			IF deviceAddrIsValid
			THEN
				Busy										:= TRUE;
				Done										:= FALSE;
				Error										:= FALSE;
				ErrorId 									:= 0;
				ErrorText									:= '';
				state										:= 1001;
			ELSE
				Busy										:= FALSE;
				Done										:= FALSE;
				Error										:= TRUE;
				ErrorId 									:= 24; //Invalid ads port 
				ErrorText									:= CONCAT('Error read parameter in state:' , TO_STRING(state * -1));
				ErrorText									:= CONCAT(ErrorText , '| ID/Addr. of device invalid');
				state										:= 9999;			
			END_IF
		ELSE                        						
			Busy											:= FALSE;
			Done											:= FALSE;
			Error											:= FALSE;
			ErrorId 										:= 0;
			ErrorText										:= '';
		END_IF

	1..99,1001..1099: (* Call sequence read *)
		IF SeqRead(state)
		THEN
			state											:= 9999;	
			InitDone										:= TRUE;
			Done											:= NOT Error;
			Busy											:= FALSE;		
		END_IF
             				
	9999: (* Last state execution finished *****************************)
		IF NOT Execute 
		THEN
			Busy											:= FALSE;
			Done											:= FALSE;
			Error											:= FALSE;
			ErrorId 										:= 0;
			ErrorText										:= '';
		END_IF
		
	ELSE (* Case else *)	
		Busy												:= FALSE;
		Error												:= TRUE;
		ErrorId												:= E_AdsErr.DEVICE_INVALIDSTATE;
		ErrorText											:= CONCAT('Error read parameter; invalid state:' , TO_STRING(state));
		ErrorText											:= CONCAT(ErrorText , ' Id:');
		ErrorText											:= CONCAT(ErrorText , TO_STRING(ErrorId));
		State												:= 9999;
	END_CASE

	(* Reset state to zero if Execute is set back to false *)
	IF NOT Execute AND NOT busy
	THEN
		MemFnc												:=  -1;
		state 												:= 0;
	END_IF
	
	Read													:= Busy; //Return;
END_IF	

(****************************************************************************************************************)
END_METHOD

METHOD PROTECTED seqRead : BOOL //Return value = TRUE if execution finished 
VAR_IN_OUT
	state							:	INT;
END_VAR
CASE state OF
1,1001:
(* Example
		IF getValue(IDxGrp:= 16#5100,	IDxOffs := 16#9,	LEN := SIZEOF(uiValue),	pActValue := ADR(uiValue),  pSetValue := 0)
		THEN
			SetRefFlag :=RefFlag							:= TO_BOOL(uiValue);
		END_IF
*)
	SeqRead													:= TRUE;
ELSE
	SeqRead													:= TRUE;
END_CASE
END_METHOD

METHOD PROTECTED seqWrite : BOOL //Return value = TRUE if execution finished 
VAR_IN_OUT
	state							:	INT;
END_VAR
CASE state OF
1,1001:
(* Example 
	setValue(IDxGrp:= 16#4000,	IDxOffs := 16#102,	LEN := SIZEOF(SetDec), pActValue := ADR(Dec),	pSetValue := ADR(SetDec));
*)
	SeqWrite												:= TRUE;
ELSE
	SeqWrite												:= TRUE;
END_CASE
END_METHOD

METHOD PUBLIC FINAL write : BOOL //Return value = TRUE if busy
VAR_INPUT
	Execute													:	BOOL;
END_VAR
IF MemFnc = FNC_READ AND busy
THEN
	Busy													:= FALSE;
	Error													:= TRUE;
	ErrorId													:= E_AdsErr.DEVICE_BUSY;
	ErrorText												:= CONCAT('Error write parameter in state:' , TO_STRING(state * -1));
	ErrorText												:= CONCAT(ErrorText , ' read parameter is active, Id:');
	ErrorText												:= CONCAT(ErrorText , TO_STRING(ErrorId));
	MemFnc													:=  -1;
	Write													:= FALSE;
ELSE
	MemFnc													:= FNC_WRITE;
	THIS^.Execute											:= Execute;

(* Parameter schreiben ************************************************************************************************)
	(* Parameter schreiben Statemaschine *)
	CASE state OF
	0:	(* Init *)	
		IF Execute 
		THEN
			IF deviceAddrIsValid
			THEN
				Busy										:= TRUE;
				Done										:= FALSE;
				Error										:= FALSE;
				ErrorId 									:= 0;
				state										:= 1001;
			ELSE
				Busy										:= FALSE;
				Done										:= FALSE;
				Error										:= TRUE;
				ErrorId 									:= 24; //Invalid ads port 	
				ErrorText									:= CONCAT('Error write parameter in state:' , TO_STRING(state * -1));
				ErrorText									:= CONCAT(ErrorText , '| ID/Addr. of device invalid');
				state										:= 9999;			
			END_IF                  						
		ELSE 
			Busy											:= FALSE;
			Done											:= FALSE;
			Error											:= FALSE;
			ErrorId 										:= 0;
			ErrorText										:= '';
		END_IF
		
	1..99,1001..1099: (* Call sequence write *)
		IF SeqWrite(state)
		THEN
			Done											:= NOT Error;
			Busy											:= FALSE;
			state											:= 9999;			
		END_IF	
		
	9999: (* Last state execution finished *****************************)
		IF NOT Execute 
		THEN
			Busy											:= FALSE;
			Done											:= FALSE;
			Error											:= FALSE;
			ErrorId 										:= 0;
			ErrorText										:= '';
		END_IF
		
	ELSE (* Case else *)	
		Busy												:= FALSE;
		Error												:= TRUE;
		ErrorId												:= E_AdsErr.DEVICE_INVALIDSTATE;
		ErrorText											:= CONCAT('Error write parameter; invalid state:' , TO_STRING(state));
		ErrorText											:= CONCAT(ErrorText , ' Id:');
		ErrorText											:= CONCAT(ErrorText , TO_STRING(ErrorId));
		State												:= 9999;
	END_CASE

	(* Reset state to zero if Execute is set back to false *)
	IF NOT Execute AND NOT busy
	THEN
		MemFnc												:=  -1;
		state 												:= 0;
	END_IF
	
	Write													:= Busy; //Return;
END_IF
END_METHOD

END_FUNCTION_BLOCK

// POUs/IO/Drives/CoE/EL72xx/AxDriveCoE_wEvents
{attribute 'no_check'}
//Drive 
FUNCTION_BLOCK AxDriveCoE_wEvents EXTENDS AxDriveCoE   
VAR_OUTPUT CONSTANT
{attribute 'displaymode':='binary'}  
	OPTION_DISABLE_INT_LIMIT_WARNING						:	BYTE := 2#0000_0001;
{attribute 'displaymode':='binary'}  
	OPTION_DISABLE_REMOTE_CNTR_NOT_ACTIVE					:	BYTE := 2#0000_0010;	
END_VAR                  						
VAR_INPUT                           						
	EnableEvent												:	BOOL := TRUE;
	{attribute 'displaymode':='binary'}  
	Options													:	BYTE := 0;
	ConfirmTrig												:	BOOL := FALSE; (* Reset event *)
	SourceId												:	UDINT := 102200; //CoE Drive default multisource Id + Ax id
	Name													:	STRING(30) := '';
	ErrorLimitPos											:	BOOL := FALSE;
	ErrorLimitNeg											:	BOOL := FALSE;
END_VAR
VAR_IN_OUT
END_VAR
VAR_OUTPUT
	EventStatus												:	DWORD;
	NoOfActiveEvents										:	INT;
END_VAR                             						
VAR

END_VAR
VAR
(* Cache *********************************************************************)
	
(* Timer ********************************************************************************)
                                						
(* Trigger ******************************************************************************)


(* Function blocks ****************************************************************************)
	
	Event													: EventHandlingGrp10;
	EventDiagMessage										: EventHandling;

(* Dummy Speicher **********************************************************)
	i														: INT := 0 ;

END_VAR

	(* CoE Drive with diag and eventlogger implementation								*)
	(************************************************************************************)

(* call super ***********************************************************************)
	SUPER^();

(* trigger events ************************************************)
	_callEvents();

(*****************************************************************)

METHOD _callEvents : BOOL
VAR_INPUT
END_VAR
(* Check if msg activ and init some parameter ***********************)
	IF Event.no[1].Text2 <> Name AND Name <> '' OR Event.no[1].Text2 = '' AND rAxis.NcToPlc.AxisId <> 0
	THEN
		Event.no[1].Class 									:= TC2_SYSTEM.TCEVENTCLASS_STATEINFO;
		Event.no[3].Class 									:= TC2_SYSTEM.TCEVENTCLASS_WARNING;
		Event.no[4].Class 									:= TC2_SYSTEM.TCEVENTCLASS_WARNING;
		Event.no[5].Class 									:= TC2_SYSTEM.TCEVENTCLASS_STATEINFO;
		Event.no[6].Class 									:= TC2_SYSTEM.TCEVENTCLASS_STATEINFO;
		Event.no[7].Class 									:= TC2_SYSTEM.TCEVENTCLASS_STATEINFO;
		
		(* Init axisname *)
		FOR i := Event.MIN_EVENT TO Event.MAX_EVENT DO
		(*	Event.no[i].Text1								:= '';*)
			Event.no[i].Text2								:= SEL(LEN(name)>1,CONCAT('Axis id:',DWORD_TO_STRING(rAxis.NcToPlc.AxisId)),name);			
		END_FOR
		EventDiagMessage.Text2								:= Event.no[1].Text2;
	END_IF

(* workl Event Ctrl *************************************************)
	Event(
		ConfirmTrig 	:= ConfirmTrig,
		Disable			:= rAxis.NcToPlc.AxisId = 0 OR NOT EnableEvent,
		SourceId		:= SourceId + rAxis.NcToPlc.AxisId);
		

(* Event diag message ***************************************************)
	CASE ReadCoEDiagMsg.MsgSeverity OF
	0: // Info message
		EventDiagMessage.Class 								:= TCEVENTCLASS_MESSAGE;
	1: // warning
		EventDiagMessage.Class 								:= TCEVENTCLASS_WARNING;
	2: // error message
		EventDiagMessage.Class 								:= TCEVENTCLASS_ALARM;
	ELSE // unknown type
		EventDiagMessage.Class 								:= TCEVENTCLASS_NONE;
	END_CASE
				
	EventDiagMessage(
		Flag			:= state = 0 AND ReadCoEDiagMsg.TextId <> 0 AND (Status.Fault OR Status.Warning) AND NOT Event.Disable,
		ConfirmTrig 	:= ConfirmTrig OR NOT EventDiagMessage.Flag AND EventDiagMessage.State <> TCEVENTSTATE_INVALID,
		MsgId			:= ReadCoEDiagMsg.TextId,
		SourceId		:= Event.SourceId);
		
(* Event status ******************************************************)
	NoOfActiveEvents										:= Event.NoOfActiveEvents + SEL(EventDiagMessage.Status.31 , 0, 1);
 	EventStatus												:= Event.Status OR EventDiagMessage.Status;

		
(* Set events at the end to allow set to false in inherited FBs ********************)
	Event.no[1].Flag 										:= NOT Status.ReadyToSwitchOn; 
	Event.no[2].Flag 										:= Status.Fault;
	Event.no[3].Flag 										:= Status.Warning; 				
	Event.no[4].Flag 										:= Status.InternalLimitActive AND NOT Options.0;
	Event.no[5].Flag 										:= Status.SwitchOnDisabled;
	Event.no[6].Flag 										:= NOT Status.FollowCmdValue AND Status.SwitchedOn AND NOT options.1 AND NOT rAxis.Status.OpMode.SimulationAxis;
	Event.no[7].Flag 										:= BreakUnlock OR BreakUnlocked; 	
	Event.no[8].Flag 										:= ErrorLimitPos;
	Event.no[9].Flag 										:= ErrorLimitNeg;
	
(************************************************************************)
	_callEvents												:= TRUE;
(******************************************************************************)
END_METHOD

METHOD PUBLIC confirm : bool
VAR_INPUT
END_VAR
confirm 								:= Event.confirm();
END_METHOD

PROPERTY PUBLIC optDisabledRemoteCntrNotActive : BOOL
GET
optDisabledRemoteCntrNotActive := Options.1;
END_GET
SET
Options.1 := optDisabledRemoteCntrNotActive;
END_SET
END_PROPERTY

PROPERTY PUBLIC optDisableIntLimitWarning : BOOL
GET
optDisableIntLimitWarning := Options.0;
END_GET
SET
Options.0 := optDisableIntLimitWarning;
END_SET
END_PROPERTY

END_FUNCTION_BLOCK

// POUs/IO/Drives/CoE/CiA_DS402Controlword
FUNCTION_BLOCK CiA_DS402Controlword
VAR_INPUT

	SwitchOn 				: BOOL;	// BIT 0 
	EnableVoltage 			: BOOL := TRUE; // Bit 1 
	QuickStop 				: BOOL; // Bit 2 inverse signal / TRUE = RUN
	EnableOperation 		: BOOL; // Bit 3 
//	Operation mode specific Bit 4 	: BOOL; // Bit 4
//	Operation mode specific Bit 5 	: BOOL; // Bit 5
//	Operation mode specific Bit 6 	: BOOL; // Bit 6
	FaultReset 				: BOOL; // Bit 7 
//	Halt 					: BOOL; // Bit 8
//	Operation mode specific Bit 9 	: BOOL; // Bit 9
//	Reserved Bit 10 	: BOOL; // Bit 10
//	Manufacturere specific Bit 11 	: BOOL; // Bit 11
//	Manufacturere specific Bit 12 	: BOOL; // Bit 12
//	Manufacturere specific Bit 13 	: BOOL; // Bit 13
//	Manufacturere specific Bit 14 	: BOOL; // Bit 14
//	Manufacturere specific Bit 15 	: BOOL; // Bit 15	
END_VAR
VAR_OUTPUT
	Cmd					:	eCiA_DS402_CONTROL_CMD;
END_VAR
VAR
END_VAR

;

METHOD PUBLIC createControlword : UINT
VAR_INPUT
	StatusState												: eCiA_DS402_STATUS_STATE;
END_VAR
(* work local state machine for control ****************************************************)
	CASE StatusState OF
	eCiA_DS402_STATUS_STATE.NOT_READY_TO_SWITCH_ON:
		;
		
	eCiA_DS402_STATUS_STATE.SWITCH_ON_DISABLED:
		IF EnableVoltage
		THEN //back to "not ready to switch on"
			createControlword								:= TO_UINT(eCiA_DS402_CONTROL_CMD.SHUTDOWN);
		ELSE //To "Ready to switch on"
			createControlword								:= TO_UINT(eCiA_DS402_CONTROL_CMD.DISABLE_VOLTAGE);
		END_IF
		
	eCiA_DS402_STATUS_STATE.READY_TO_SWITCH_ON:
		IF NOT EnableVoltage
		THEN //Back to switched on disabled
			createControlword								:= TO_UINT(eCiA_DS402_CONTROL_CMD.DISABLE_VOLTAGE);
		ELSIF SwitchOn
		THEN //To switched on
			createControlword								:= TO_UINT(eCiA_DS402_CONTROL_CMD.SWITCH_ON);	
		END_IF	
		
	eCiA_DS402_STATUS_STATE.SWITCHED_ON:
		IF NOT SwitchOn
		THEN
			createControlword								:= TO_UINT(eCiA_DS402_CONTROL_CMD.SHUTDOWN);
		ELSIF NOT EnableVoltage
		THEN //Back to switched on disabled
			createControlword								:= TO_UINT(eCiA_DS402_CONTROL_CMD.DISABLE_VOLTAGE);
		ELSIF EnableOperation
		THEN // To operation enabled
			createControlword								:= TO_UINT(eCiA_DS402_CONTROL_CMD.ENABLE_OPERATION);										
		END_IF
		
	eCiA_DS402_STATUS_STATE.OPERATION_ENABLED:
		IF NOT EnableOperation 
		THEN //go back to switched on
			createControlword								:= TO_UINT(eCiA_DS402_CONTROL_CMD.SWITCH_ON);
		ELSIF NOT SwitchOn		
		THEN // back to ready to switch on 
			createControlword								:= TO_UINT(eCiA_DS402_CONTROL_CMD.SHUTDOWN);	 
		ELSIF QuickStop 
		THEN 
			createControlword								:= TO_UINT(eCiA_DS402_CONTROL_CMD.QUICK_STOP);
		ELSIF NOT EnableVoltage
		THEN //Back to switch on disabled
			createControlword								:= TO_UINT(eCiA_DS402_CONTROL_CMD.DISABLE_VOLTAGE);
		END_IF
		
	eCiA_DS402_STATUS_STATE.QUICK_STOP_ACTIVE:
		;
		
	eCiA_DS402_STATUS_STATE.FAULT_ACTIVE:
		IF NOT EnableVoltage
		THEN //back to "not ready to switch on"
			createControlword								:= TO_UINT(eCiA_DS402_CONTROL_CMD.DISABLE_VOLTAGE);
		ELSE //To "Ready to switch on"
			createControlword								:= TO_UINT(eCiA_DS402_CONTROL_CMD.SHUTDOWN);
		END_IF
		
	eCiA_DS402_STATUS_STATE.FAULT_REACTION_ACTIVE:
		;		
	END_CASE
	
(* Write controlword ********************************************************)
	Cmd													:= TO_INT(createControlword);
	createControlword.7										:= FaultReset; 
	
(*****************************************************************************)
END_METHOD

END_FUNCTION_BLOCK

// POUs/IO/Drives/DC/Ey73xx/AxDriveDC
{attribute 'no_check'}
//Beckhoff Stepper terminal status and diagnoses/ EP Box used with NC axis
//EventHandling instance use inside
FUNCTION_BLOCK AxDriveDC EXTENDS AxDriveBase
VAR CONSTANT         	
END_VAR  
VAR_INPUT
END_VAR                     					
VAR_IN_OUT                  					
END_VAR                     					
VAR_OUTPUT                  					
	Status_ReadyToEnable									: BOOL;
	Status_Ready											: BOOL;
	Status_Warning											: BOOL;
	Status_Error											: BOOL;
	Status_MovingPos										: BOOL;
	Status_MovingNeg										: BOOL;
	Status_TorqueReduced									: BOOL;
	Status_DigInput1										: BOOL;
	Status_DigInput2										: BOOL;
	Status_SyncError										: BOOL;
	Status_TxPDOToggle										: BOOL;
	InfoData1										AT %I*	:	UINT;
	InfoData2										AT %I*	:	UINT;
END_VAR                     					                   					
VAR                         					
END_VAR
VAR

(* Cache *********************************************************************)
	StatusTrig												:	BYTE;
	MemStatusTrig											:	BYTE;
	MemCoeCache												: 	ARRAY[0..5] OF BYTE; //Index A020/A030 with a lenght of 17 subindex	
	
//Diag read by CoE
	Diag_Saturated											: BOOL; // Driver stage operates with maximum duty cycle
	Diag_OverTemperature 									: BOOL; // Internal terminal temperature is higher than 80°C (see subindex 0xF80F:04)
	Diag_TorqueOverloaded 									: BOOL; // Motor current is higher than the rated current
	Diag_UnderVoltage 										: BOOL; // Motor supply voltage is 20% lower than the configured nominal voltage
	Diag_OverVoltage 										: BOOL; // Motor supply voltage is 10% higher than the configured nominal voltage
	Diag_ShortCircuit 										: BOOL; // Short circuit 
	Diag_ShortCircuitB										: BOOL; // Short circuit
	Diag_NoControlPower 									: BOOL; // Control voltage at the power contacts is less than 12 V
	Diag_MiscError 											: BOOL; // Terminal initialization failed, or supply voltage is less than 8 V, or internal terminal temperature is higher than 100°C (see subindex 0xF80F:05)
	Diag_Configuration 										: BOOL; // CoE change has not yet been adopted into the current configuration
	Diag_MotorStall											: BOOL; // A loss of step has occurred
	Diag_OpenLoadA											: BOOL; // Open load on coil A - e.g. no motor connected
	Diag_OpenLoadB											: BOOL; // Open load on coil B - e.g. no motor connected

	Diag_ActualMode											: BYTE; // Current operating mode (relevant for activated automatic mode, see 0x8012:01)
	
(* Timer ********************************************************************************)

(* Trigger ******************************************************************************)

(* Instance ****************************************************************************)
	CoERead													:	FB_EcCoeSdoReadEx := (tTimeout := DEFAULT_ADS_TIMEOUT);	//Read data via CoE
	
(* Dummy Speicher **********************************************************)
END_VAR

	(* DC Drive Control															*)
	(************************************************************************************)

(* abort function-call if the reference is invalid *****************************)
IF NOT __ISVALIDREF(rAxis) 
THEN
	Fault													:= TRUE;
	SwitchedOn												:= FALSE;
	Ready													:= FALSE;
	RETURN;
END_IF

(* Call super class ****************************************************)
	SUPER^(); 

(* Read Statusword ********************************************************)
	Status_ReadyToEnable									:= StatusWord.0 OR rAxis.Status.OpMode.SimulationAxis ;
	Status_Ready											:= StatusWord.1 OR rAxis.Status.OpMode.SimulationAxis;
	Status_Warning											:= StatusWord.2;
	Status_Error											:= StatusWord.3;
	Status_MovingPos										:= StatusWord.4;
	Status_MovingNeg										:= StatusWord.5;
	Status_TorqueReduced									:= StatusWord.6;              
             					   
	Status_DigInput1										:= StatusWord.11;
	Status_DigInput2										:= StatusWord.12;
	Status_SyncError										:= StatusWord.13;
//	_StatusWord.14;//6                                         
	Status_TxPDOToggle										:= StatusWord.15;

(* Read diag data ************************************************)
	StatusTrig.0											:= NOT Status_ReadyToEnable;
	StatusTrig.1											:= Status_Error;
	StatusTrig.2											:= Status_Warning;
	
	CASE state OF
	0:
		IF StatusTrig <> MemStatusTrig AND NOT rAxis.Status.OpMode.SimulationAxis AND AdsAddr.port > 0 
		THEN
			CoERead(
				sNetId		:= F_CreateAmsNetId(nIds :=AdsAddr.netId), 
				nSlaveAddr	:= AdsAddr.port, 
				nSubIndex	:= , 
				nIndex		:= , 
				pDstBuf		:= , 
				cbBufLen	:= , 
				bExecute	:= FALSE,
				bCompleteAccess:= TRUE, 
				tTimeout	:= , 
				bBusy		=> , 
				bError		=> , 
				nErrId		=> );
			IF NOT CoERead.bBusy
			THEN
				MemStatusTrig 								:= StatusTrig;			
				state 										:= state + 1;
			END_IF
		END_IF
	1: 
		CoERead(
			bExecute	:= TRUE, 
			nIndex		:= SEL(Channel=0,16#A030,16#A020),
			nSubIndex	:= 16#0, 
			pDstBuf		:= ADR(MemCoeCache), 
			cbBufLen	:= SIZEOF(MemCoeCache));
		IF NOT CoERead.bBusy
		THEN
			IF CoERead.bError
			THEN
				state 										:= 0;
			ELSE
				//											:= MemCoeChache[0]; 	//Subindex 0x00 Maximal sub index
				//											:= MemCoeChache[1];		//reserved				
				Diag_Saturated								:= MemCoeCache[2].0; 	//Subindex 0x01 
				Diag_OverTemperature 						:= MemCoeCache[2].1; 	//Subindex 0x02 
				Diag_TorqueOverloaded 						:= MemCoeCache[2].2; 	//Subindex 0x03 
				Diag_UnderVoltage 							:= MemCoeCache[2].3; 	//Subindex 0x04 
				Diag_OverVoltage 							:= MemCoeCache[2].4; 	//Subindex 0x05 
				Diag_ShortCircuit 							:= MemCoeCache[2].5; 	//Subindex 0x06   
				Diag_NoControlPower 						:= MemCoeCache[2].7; 	//Subindex 0x08 
				Diag_MiscError 								:= MemCoeCache[3].0; 	//Subindex 0x09
				Diag_Configuration 							:= MemCoeCache[3].1; 	//Subindex 0x0A
				//											:= MemCoeCache[3].2; 	//Subindex 0x0B 
				//											:= MemCoeCache[3].3; 	//Subindex 0x0C 
				//	 										:= MemCoeCache[3].4; 	//Subindex 0x0D 
				//				 							:= MemCoeChache[3].5; 	//Subindex 0x0E 
				//				 							:= MemCoeChache[3].6; 	//Subindex 0x0F 
				//				 							:= MemCoeChache[3].7; 	//Subindex 0x10 								
				Diag_ActualMode	 							:= MemCoeCache[4]; 	//Subindex 0x11 (e.g. 17) 
				//				 							:= MemCoeChache[5];		//reserved
	
				state										:= 0;			
			END_IF
			CoERead(bExecute := False);		
		END_IF
	END_CASE
	
(* DriveStatusBits ***********************************************)
	Fault													:= Status_Error
															//	OR Status_MotorStall
																OR Status_SyncError
																OR rAxis.NcToPlc.StateDWord.28 (* DriveDeviceError *)
																OR rAxis.NcToPlc.StateDWord.30; (* IODataInvalid *)
         											
													
	Ready	 												:= NOT Fault
																AND(Status_ReadyToEnable OR Status_Ready);
	SwitchedOn												:= Status_Ready AND NOT Fault;
	
(*******************************************************************)

END_FUNCTION_BLOCK

// POUs/IO/Drives/DC/Ey73xx/AxDriveDC_wEvents
{attribute 'no_check'}
//Beckhoff Stepper terminal diag and diagnosis with eventlogger - extended from AxDriveStepper
//EventHandling instance use inside
FUNCTION_BLOCK AxDriveDC_wEvents EXTENDS AxDriveDC
VAR CONSTANT         	
END_VAR  
VAR_INPUT
	EnableEvent												:	BOOL := TRUE; //Enable to show events
	ConfirmTrig												:	BOOL := FALSE; //Quit events
	SourceId												:	UDINT := 102700; //CoE / MDP733 DC-Motor Drive (EL73xx) default multisource Id + Ax id
	Name													:	STRING(30) := '';
	ErrorLimitPos											:	BOOL := FALSE;
	ErrorLimitNeg											:	BOOL := FALSE;
END_VAR                     					
VAR_IN_OUT                  					
END_VAR                     					
VAR_OUTPUT                  					
 	EventStatus												:	DWORD;       
	NoOfActiveEvents										:	INT;                    					
END_VAR                     					                   					
VAR                         					
END_VAR
VAR

(* Cache *********************************************************************)
	
(* Timer ********************************************************************************)

(* Trigger ******************************************************************************)

(* Instance ****************************************************************************)
	Event													:	EventHandlingGrp10;
	
(* Dummy Speicher **********************************************************)
	i														: INT := 0 ;
END_VAR

	(* Stepper Drive Control with events												*)
	(************************************************************************************)

(* Call super **********************************************)
	SUPER^();
	
(* work events *******************************************)
	_callEvents();

(*******************************************************)

METHOD PRIVATE _callEvents : BOOL
VAR_INPUT
END_VAR

(* Check if msg activ and init some parameter ***********************)
	IF Event.no[1].Text2 <> Name AND Name <> '' OR Event.no[1].Text2 = '' AND rAxis.NcToPlc.AxisId <> 0
	THEN
		Event.no[1].Class 									:= TC2_SYSTEM.TCEVENTCLASS_STATEINFO;
		Event.no[3].Class 									:= TC2_SYSTEM.TCEVENTCLASS_WARNING;
		
		(* Init Achsname *)
		FOR i := Event.MIN_EVENT TO Event.MAX_EVENT DO
		(*	Event.no[i].Text1								:= '';*)
			Event.no[i].Text2								:= SEL(LEN(name)>1,CONCAT('Axis id:',DWORD_TO_STRING(rAxis.NcToPlc.AxisId)),name);
		END_FOR
	END_IF

(* workl Event Ctrl *************************************************)
	Event(
		ConfirmTrig := ConfirmTrig,
		Disable		:= rAxis.NcToPlc.AxisId = 0 OR NOT EnableEvent,
		SourceId	:= SourceId + rAxis.NcToPlc.AxisId,
		Status		=> EventStatus,
		NoOfActiveEvents => NoOfActiveEvents);

(* Event Logger Meldungen *****************************************************)
	Event.no[1].Flag 										:= NOT Status_ReadyToEnable ; 
	Event.no[2].Flag 										:= Fault;
	Event.no[3].Flag 										:= (Status_Warning OR Diag_Configuration) AND NOT rAxis.Status.Homing AND NOT rAxis.Status.Disabled; //Avoid warning if drive is disabled (EL7037 and older FB on EL7047 - 2020-03-26) 				
	Event.no[4].Flag 										:= Diag_TorqueOverloaded;
	Event.no[5].Flag 										:= Diag_UnderVoltage OR Diag_OverVoltage OR Diag_NoControlPower;
	Event.no[6].Flag 										:= Diag_ShortCircuit;
	Event.no[7].Flag 										:= Diag_Saturated;
	Event.no[8].Flag										:= Diag_OverTemperature ;
	Event.no[9].Flag 										:= ErrorLimitPos; 	
	Event.no[10].Flag 										:= ErrorLimitNeg;	
(*	Event.no[11].Flag 										:= FALSE; 				
	Event.no[12].Flag 										:= FALSE;					
	Event.no[13].Flag 										:= FALSE; 			Event.no[9].Class := TC2_SYSTEM.TCEVENTCLASS_WARNING;
	Event.no[14].Flag 										:= FALSE; 			Event.no[10].Class := TC2_SYSTEM.TCEVENTCLASS_WARNING;
	Event.no[15].Flag 										:= FALSE;
	Event.no[16].Flag 										:= FALSE;
	Event.no[17].Flag 										:= FALSE;
	Event.no[18].Flag 										:= FALSE;
	Event.no[19].Flag 										:= FALSE;
	Event.no[20].Flag 										:= FALSE;
	Event.no[21].Flag 										:= FALSE;
	Event.no[22].Flag 										:= FALSE;
	Event.no[23].Flag 										:= FALSE;
	Event.no[24].Flag 										:= FALSE;
	Event.no[25].Flag 										:= FALSE;
*)

(******************************************************************************)
END_METHOD

METHOD PUBLIC confirm : bool
VAR_INPUT
END_VAR
confirm			:= Event.confirm();
END_METHOD

END_FUNCTION_BLOCK

// POUs/IO/Drives/Stepper/AxDriveStepper
{attribute 'no_check'}
//Beckhoff Stepper terminal status and diagnoses/ EP Box used with NC axis
//EventHandling instance use inside
FUNCTION_BLOCK AxDriveStepper EXTENDS AxDriveBase
VAR CONSTANT         	
END_VAR  
VAR_INPUT
END_VAR                     					
VAR_IN_OUT                  					
END_VAR                     					
VAR_OUTPUT                  					
	Status_ReadyToEnable									: BOOL;
	Status_Ready											: BOOL;
	Status_Warning											: BOOL;
	Status_Error											: BOOL;
	Status_MovingPos										: BOOL;
	Status_MovingNeg										: BOOL;
	Status_TorqueReduced									: BOOL;
	Status_MotorStall										: BOOL;
	Status_DigInput1										: BOOL;
	Status_DigInput2										: BOOL;
	Status_SyncError										: BOOL;
	Status_TxPDOToggle										: BOOL;
	InfoData1										AT %I*	:	UINT;
	InfoData2										AT %I*	:	UINT;
END_VAR                     					                   					
VAR                         					
END_VAR
VAR

(* Cache *********************************************************************)
	StatusTrig												:	BYTE;
	MemStatusTrig											:	BYTE;
	MemCoeCache											: 	ARRAY[0..5] OF BYTE; //Index A010 with a lenght of 17 subindex	
	
//Diag read by CoE
	Diag_Saturated											: BOOL; // Driver stage operates with maximum duty cycle
	Diag_OverTemperature 									: BOOL; // Internal terminal temperature is higher than 80°C (see subindex 0xF80F:04)
	Diag_TorqueOverloaded 									: BOOL; // Motor current is higher than the rated current
	Diag_UnderVoltage 										: BOOL; // Motor supply voltage is 20% lower than the configured nominal voltage
	Diag_OverVoltage 										: BOOL; // Motor supply voltage is 10% higher than the configured nominal voltage
	Diag_ShortCircuit 										: BOOL; // Short circuit 
	Diag_ShortCircuitB										: BOOL; // Short circuit
	Diag_NoControlPower 									: BOOL; // Control voltage at the power contacts is less than 12 V
	Diag_MiscError 											: BOOL; // Terminal initialization failed, or supply voltage is less than 8 V, or internal terminal temperature is higher than 100°C (see subindex 0xF80F:05)
	Diag_Configuration 										: BOOL; // CoE change has not yet been adopted into the current configuration
	Diag_MotorStall											: BOOL; // A loss of step has occurred
	Diag_OpenLoadA											: BOOL; // Open load on coil A - e.g. no motor connected
	Diag_OpenLoadB											: BOOL; // Open load on coil B - e.g. no motor connected

	Diag_ActualMode											: BYTE; // Current operating mode (relevant for activated automatic mode, see 0x8012:01)
	
(* Timer ********************************************************************************)

(* Trigger ******************************************************************************)

(* Instance ****************************************************************************)
	CoERead													:	FB_EcCoeSdoReadEx := (tTimeout := DEFAULT_ADS_TIMEOUT);	//Read data via CoE
	
(* Dummy Speicher **********************************************************)
END_VAR

	(* Stepper Drive Control															*)
	(************************************************************************************)

(* abort function-call if the reference is invalid *****************************)
IF NOT __ISVALIDREF(rAxis) 
THEN
	Fault													:= TRUE;
	SwitchedOn												:= FALSE;
	Ready													:= FALSE;
	RETURN;
END_IF

(* Call super class ****************************************************)
	SUPER^();
	
(* Read Statusword ********************************************************)
	Status_ReadyToEnable									:= StatusWord.0 OR rAxis.Status.OpMode.SimulationAxis ;
	Status_Ready											:= StatusWord.1 OR rAxis.Status.OpMode.SimulationAxis;
	Status_Warning											:= StatusWord.2;
	Status_Error											:= StatusWord.3;
	Status_MovingPos										:= StatusWord.4;
	Status_MovingNeg										:= StatusWord.5;
	Status_TorqueReduced									:= StatusWord.6;
	Status_MotorStall										:= StatusWord.7;
//	_StatusWord.8; //0                  					   
//	_StatusWord.9; //1                  					   
//	_StatusWord.10;//2                  					   
	Status_DigInput1										:= StatusWord.11;
	Status_DigInput2										:= StatusWord.12;
	Status_SyncError										:= StatusWord.13;
//	_StatusWord.14;//6                                         
	Status_TxPDOToggle										:= StatusWord.15;

(* Read diag data ************************************************)
	StatusTrig.0											:= NOT Status_ReadyToEnable;
	StatusTrig.1											:= Status_Error;
	StatusTrig.2											:= Status_Warning;
	
	CASE state OF
	0:
		IF StatusTrig <> MemStatusTrig AND NOT rAxis.Status.OpMode.SimulationAxis AND AdsAddr.port > 0 
		THEN
			CoERead(
				sNetId		:= F_CreateAmsNetId(nIds :=AdsAddr.netId), 
				nSlaveAddr	:= AdsAddr.port, 
				nSubIndex	:= , 
				nIndex		:= , 
				pDstBuf		:= , 
				cbBufLen	:= , 
				bExecute	:= FALSE,
				bCompleteAccess:= TRUE, 
				tTimeout	:= , 
				bBusy		=> , 
				bError		=> , 
				nErrId		=> );
			IF NOT CoERead.bBusy
			THEN
				MemStatusTrig 								:= StatusTrig;			
				state 										:= state + 1;
			END_IF
		END_IF
	1: 
		CoERead(
			bExecute	:= TRUE, 
			nIndex		:= 16#A010,
			nSubIndex	:= 16#0, 
			pDstBuf		:= ADR(MemCoeCache), 
			cbBufLen	:= SIZEOF(MemCoeCache));
		IF NOT CoERead.bBusy
		THEN
			IF CoERead.bError
			THEN
				state 										:= 0;
			ELSE
				//											:= MemCoeChache[0]; 	//Subindex 0x00 Maximal sub index
				//											:= MemCoeChache[1];		//reserved				
				Diag_Saturated								:= MemCoeCache[2].0; 	//Subindex 0x01 
				Diag_OverTemperature 						:= MemCoeCache[2].1; 	//Subindex 0x02 
				Diag_TorqueOverloaded 						:= MemCoeCache[2].2; 	//Subindex 0x03 
				Diag_UnderVoltage 							:= MemCoeCache[2].3; 	//Subindex 0x04 
				Diag_OverVoltage 							:= MemCoeCache[2].4; 	//Subindex 0x05 
				Diag_ShortCircuit 							:= MemCoeCache[2].5; 	//Subindex 0x06   
				Diag_ShortCircuitB 							:= MemCoeCache[2].6; 	//Subindex 0x07 - only at EL70x1
				Diag_NoControlPower 						:= MemCoeCache[2].7; 	//Subindex 0x08 
				Diag_MiscError 								:= MemCoeCache[3].0; 	//Subindex 0x09
				Diag_Configuration 							:= MemCoeCache[3].1; 	//Subindex 0x0A
				Diag_MotorStall 							:= MemCoeCache[3].2; 	//Subindex 0x0B 
				Diag_OpenLoadA 								:= MemCoeCache[3].3; 	//Subindex 0x0C 
				Diag_OpenLoadB	 							:= MemCoeCache[3].4; 	//Subindex 0x0D 
				//				 							:= MemCoeChache[3].5; 	//Subindex 0x0E 
				//				 							:= MemCoeChache[3].6; 	//Subindex 0x0F 
				//				 							:= MemCoeChache[3].7; 	//Subindex 0x10 								
				Diag_ActualMode	 							:= MemCoeCache[4]; 	//Subindex 0x11 (e.g. 17) 
				//				 							:= MemCoeChache[5];		//reserved
	
				state										:= 0;			
			END_IF
			CoERead(bExecute := False);		
		END_IF
	END_CASE
	
(* DriveStatusBits ***********************************************)
	Fault													:= Status_Error
															//	OR Status_MotorStall
																OR Status_SyncError
																OR rAxis.NcToPlc.StateDWord.28 (* DriveDeviceError *)
																OR rAxis.NcToPlc.StateDWord.30; (* IODataInvalid *)
         											
													
	Ready	 												:= NOT Fault
																AND(Status_ReadyToEnable OR Status_Ready);
	SwitchedOn												:= Status_Ready AND NOT Fault;
	
(*******************************************************************)

END_FUNCTION_BLOCK

// POUs/IO/Drives/SoE/Ax580x
{attribute 'no_check'}
//AX5000 safety card option IOs - AX5805/AX5806 FSoE slave inputs 
FUNCTION_BLOCK Ax580x 
VAR_INPUT
END_VAR
VAR_OUTPUT
	STO												AT %I*		:	BOOL;	//option Safe Torque Off
	SSM_1											AT %I*		:	BOOL;	//option Safe Speed Monitor 1
	SSM_2											AT %I*		:	BOOL;	//option Safe Speed Monitor 2
	SOS_1											AT %I*		:	BOOL;	//option Safe Operating Speed 1
	SSR_1											AT %I*		:	BOOL;	//option Safe Speed Range 1
	SDIp											AT %I*		:	BOOL;	//option Safe Direction positive
	SDIn											AT %I*		:	BOOL;	//option Safe Direction negative
	Error											AT %I*		:	BOOL;	//Error active or error ack 
	SLS_1											AT %I*		:	BOOL;	//special config (Safe Limited Speed)
	
	PositionActualValue								AT %I*	:	DINT;		//contains actual position value of drive 
	VelocityActualValue								AT %I*	:	DINT;		//contains actual velocity value of drive	
END_VAR         								
VAR             								
END_VAR

(* AX5805/06 AX5000 servo drives safety card FSoE slave inputs		*)
(********************************************************************)

(* Input Signals Valid ******************************************************)
(* not in use
	STO														:= SafeDataByte.0;
	SSM_1													:= SafeDataByte.1;
	SSM_2													:= SafeDataByte.2;
	SOS_1													:= SafeDataByte.3;
	SSR_1													:= SafeDataByte.4;
	SDIp													:= SafeDataByte.5;
	SDIn													:= SafeDataByte.6;
	Error													:= SafeDataByte.7;
	SLS_1													:= SafeDataByte.8; // Special Config
*)
(**********************************************************************)

END_FUNCTION_BLOCK

// POUs/IO/Drives/SoE/AxDriveSoE_Ax5000
{attribute 'no_check'}
//AX5000 SoE drive status and diagnosis FB
FUNCTION_BLOCK AxDriveSoE_Ax5000 extends AxDriveBase (* Lips: TcMc2Drive, TcDrive *)
VAR_INPUT
	ResetTrig												:	BOOL;
	BreakUnlock												:	BOOL;
	BreakLock												:	BOOL;					
END_VAR                 									
VAR_IN_OUT              									
END_VAR                 									
VAR_OUTPUT              	                    										
	BreakStatus												:	BOOL; (* FALSE = ON / TRUE = OFF *)                        								
	RT_StatusChanged										:	BOOL;
{attribute 'displaymode':='binary'}
	MotorsStatusWord										:	WORD; 
	Status													:	ST_AX5000DriveStatus;
	C1D														:	ST_AX5000_C1D;
	DiagMsg 												: 	ST_SoE_String;
	DiagNumber 												: 	UDINT;
	SafetyError										AT %I*	:	BOOL;	(* Ax5805 Drive Safety Error - Bit .7 in Input Safe Data Byte 0 oder 2 *)	
	SercosErrorId											:	UINT;
END_VAR
VAR_OUTPUT CONSTANT
END_VAR
VAR (* EA Internal *)
	(* P-0-0205 - muss ins Zyklische Interface des Reglers unter S-0-0016 (AT) gemappt,
		und dann direkt mit der PLC-Variable verknüpft werden. 
		Oder für das Lesen auf Anforderung die Deklaration auf Lokale Variable ändern 
		und in der Statemaschine für das Status lesen 
		den Auskommentierten Teil mit ins Programm nehmen 
	*)
(*	PwrMgmStatusWord AT %I* : WORD; *)
(*	PwrMgmStatusWord : WORD; *)

END_VAR
VAR

(* Zwischenspeicher *********************************************************************)
	MemDriveStatusword										: 	WORD;
	
	MEM_StatusTrig											:	BYTE;
	StatusTrig												:	BYTE;
	stateReadStatus											:	INT;

(* Timer ********************************************************************************)

(* Trigger ******************************************************************************)

(* Bausteine ****************************************************************************)
	SoEAX5000SetMotorCtrlWord 								: FB_SoEAX5000SetMotorCtrlWord_ByDriveRef := (tTimeout := DEFAULT_ADS_TIMEOUT);	(* Bremse manuell lösen *)
	SoEDriveReset											: FB_SoEReset_ByDriveRef := (tTimeout	:= DEFAULT_ADS_TIMEOUT);
	SoERead													: FB_SoERead_ByDriveRef := (tTimeout:= DEFAULT_ADS_TIMEOUT);

(* Dummy Speicher **********************************************************)
	_WORD													: WORD;
(****************************************************************************)
END_VAR

	(************************************************************************************)
	(*																					*)
	(*		B E C K H O F F   N E W   A U T O M A T I O N   T E C H N O L O G Y    		*)
	(*																					*)
	(*		Eiserstr.5	D-33415 Verl	Germany	phone:	+49-5246-0	www.Beckhoff.Com	*)
    (*																					*)
    (*		Bausteinbeschreibung	:	AX5000 Drive Ctrl								*)
	(*		TwinCAT-Version			:	3.x or higher 									*)
	(*		Version					:	V3.0 											*)
 	(*		Autor					:	Daniel Schlingmann								*)
	(*		Lib						:	TcMc2Drive.lib / TcDrive.Lib					*)
	(*																					*)
	(************************************************************************************)

(* abort function-call if the reference is invalid *****************************)
IF NOT __ISVALIDREF(rAxis)  THEN
	Fault													:= TRUE;
	Ready													:= FALSE;
	SwitchedOn												:= FALSE;
	RETURN;
END_IF

(* Call super class ****************************************************)
	SUPER^(); 
	
(* DriveStatusword *****************************)
	Status 													:= F_ConvWordToSTAX5000DriveStatus(StatusWord);
	IF rAxis.Status.OpMode.SimulationAxis OR AdsAddr.port = 0
	THEN
		Status.bNotReadyToPowerUp							:= FALSE;	
		Status.bDrvShutdownBitC1D							:= FALSE;
		Status.bReadyForEnable								:= TRUE;
		Status.bEnabled										:= TRUE;	
	END_IF
	(* PowerManagementStatusWord Auswerten *)
	(* Bit 0 = Status UMain ok, ok = True
		Bit 1 = Umain Overvoltage, active = True
		Bit 2 = Umain phase error, error = False
		Bit 3 = Status DcLink ok, ok = True
		Bit 4 = Ext. Umain relay, ready to Switch on = True
		Bit 5 = Status Fan, aktive = True 
		Bit 6 = Status load relay, active = True
		Bit 7 = Status internal chopper, active = True
		Bit 8 = Status external chopper, active = True
		Bit 9 = Status additinal fan, active = True
		Bit 10-15 = reserved *)
	(*
	ReadyForContactor := PowerManagementStatusWord.4;
	*)

(* DriveStatusBits ***********************************************)
	Fault													:= Status.bDrvShutdownBitC1D
																OR rAxis.NcToPlc.StateDWord.28 (* DriveDeviceError *)
																OR rAxis.NcToPlc.StateDWord.30 (* IODataInvalid *)
																OR SafetyError;
            												
	Ready 													:= NOT Fault
																AND(Status.bReadyForEnable OR Status.bEnabled)
																(* AND ReadyForContactor AX 5000 *);

	SwitchedOn												:= Status.bEnabled AND NOT Fault;	
																
(* Init drive ref *************************************************)
	IF AdsAddr.port <> SoEDriveReset.stDriveRef.nSlaveAddr 
	THEN
		SoEDriveReset.stDriveRef.sNetId						:= F_CreateAmsNetId(AdsAddr.netId);	
		SoEDriveReset.stDriveRef.nSlaveAddr					:= AdsAddr.port;	
		SoEDriveReset.stDriveRef.nDriveNo					:= Channel;	
		
		SoEAX5000SetMotorCtrlWord.stDriveRef				:= 	
		SoERead.stDriveRef		 							:= SoEDriveReset.stDriveRef;
	END_IF

(* Reset Drive ****************************************************)
	SoEDriveReset();
	IF SoEDriveReset.bBusy 
	THEN
		; (* Block ist currend working *)
	ELSIF ResetTrig
	THEN
		reset();
	ELSIF SoEDriveReset.bExecute
	THEN
		RefreshStatus();
		SoEDriveReset.bExecute 								:= FALSE;
	END_IF

(* Bremse loesen/setzen  ***********************************************)
	IF (SoEAX5000SetMotorCtrlWord.bForceUnLock XOR BreakUnlock)
		OR (SoEAX5000SetMotorCtrlWord.bForceLock XOR Breaklock)
		OR SoEAX5000SetMotorCtrlWord.bBusy 
	THEN
		SoEAX5000SetMotorCtrlWord(
			stDriveRef	:= ,  //See above
			bExecute	:= NOT SoEAX5000SetMotorCtrlWord.bBusy AND NOT rAxis.Status.OpMode.SimulationAxis, 
			tTimeout	:= , 
			bForceLock	:= Breaklock , 
			bForceUnlock:= BreakUnlock , 
			bBusy		=> , 
			bError		=>  , 
			iAdsErrId	=> , 
			iSercosErrId=> );
	END_IF

(* DriveStatusword auswerten Sercos *****************************)
	RT_StatusChanged 										:= SHR(StatusWord,2) <> MemDriveStatusword;
	MemDriveStatusword 										:= SHR(StatusWord,2);

(* Start Read Drive status *****************************************************************)
	CASE stateReadStatus OF
	0:
		StatusTrig.0 										:= rAxis.NcToPlc.StateDWord.28;
		StatusTrig.1 										:= rAxis.NcToPlc.StateDWord.30;

		IF NOT rAxis.Status.OpMode.SimulationAxis AND AdsAddr.port > 0
			AND(RT_StatusChanged OR MEM_StatusTrig <> StatusTrig)
		THEN
			RefreshStatus();
		ELSE
			;
		END_IF

	(* Read Class 1 Diag *********************************************************)
	10:
		IF NOT SoERead.bBusy
			AND SoERead.bExecute
		THEN
			IF SoERead.bError THEN
				stateReadStatus 							:= 0;
			ELSE                        					
				C1D 										:= F_ConvWordToSTAX5000C1D(_WORD);
				stateReadStatus 							:= stateReadStatus + 1;
			END_IF
		END_IF

		SoERead(
			stDriveRef	:= ,  //See init for drive ref
			nIdn		:= S_0_IDN + 11,
			nElement	:= EC_SOE_ELEMENT_VALUE (* 16#40*),
			pDstBuf		:= ADR(_WORD),
			cbBufLen	:= SIZEOF(_WORD),
			bExecute	:= stateReadStatus = 10,
			tTimeout	:= ,
			bBusy		=> ,
			bError		=> ,
			iAdsErrId	=> ,
			iSercosErrId=> ,
			dwAttribute	=> );

	(* Motor Statusword ***************************************************)
	11:
		IF NOT SoERead.bBusy
			AND SoERead.bExecute
		THEN
			IF SoERead.bError 
			THEN
				stateReadStatus 							:= 0;
			ELSE
				BreakStatus 								:= MotorsStatusWord.0;
				stateReadStatus 							:= stateReadStatus + 1;
			END_IF
		END_IF

		SoERead(
			stDriveRef	:= ,  //See init for drive ref
			nIdn		:= P_0_IDN + 97, (* Motor Status word *)
			nElement	:= EC_SOE_ELEMENT_VALUE (* 16#40*),
			pDstBuf		:= ADR(MotorsStatusWord),
			cbBufLen	:= SIZEOF(MotorsStatusWord),
			bExecute	:= stateReadStatus = 11,
			tTimeout	:= ,
			bBusy		=> ,
			bError		=> ,
			iAdsErrId	=> ,
			iSercosErrId=> ,
			dwAttribute	=> );


	(* Diag Message *********************************************************)
	12:
		IF NOT SoERead.bBusy
			AND SoERead.bExecute
		THEN
			IF SoERead.bError 
			THEN
				stateReadStatus 							:= 0;
			ELSE
				stateReadStatus 							:= stateReadStatus + 1;
			END_IF
		END_IF

		SoERead(
			stDriveRef	:= ,  //See init for drive ref
			nIdn		:= S_0_IDN + 95,
			nElement	:= EC_SOE_ELEMENT_VALUE (* 16#40*),
			pDstBuf		:= ADR(DiagMsg),
			cbBufLen	:= SIZEOF(DiagMsg),
			bExecute	:= stateReadStatus = 12,
			tTimeout	:= ,
			bBusy		=> ,
			bError		=> ,
			iAdsErrId	=> ,
			iSercosErrId=> ,
			dwAttribute	=> );

	(* Diag Number *********************************************************)
	13:
		IF NOT SoERead.bBusy
			AND SoERead.bExecute
		THEN
			IF SoERead.bError 
			THEN
				stateReadStatus 							:= 0;
			ELSE
				stateReadStatus 							:= stateReadStatus + 1;
			END_IF
		END_IF
		
		SoERead(
			stDriveRef	:= ,  //See init for drive ref
			nIdn		:= S_0_IDN + 390,
			nElement	:= EC_SOE_ELEMENT_VALUE (* 16#40*),
			pDstBuf		:= ADR(DiagNumber),
			cbBufLen	:= SIZEOF(DiagNumber),
			bExecute	:= stateReadStatus = 13,
			tTimeout	:= ,
			bBusy		=> ,
			bError		=> ,
			iAdsErrId	=> ,
			iSercosErrId=> ,
			dwAttribute	=> );

	(* reading status finished ************************************************************)
	ELSE (* Case else *)
		stateReadStatus 									:= 0;
	END_CASE

(******************************************************************************************)

METHOD PUBLIC break : BOOL //Return value = TRUE if busy
VAR_INPUT
	lock													: BOOL;
END_VAR
BreakLock													:= lock AND NOT rAxis.Status.OpMode.SimulationAxis;
BreakUnlock													:= NOT lock AND NOT rAxis.Status.OpMode.SimulationAxis;
break														:= (SoEAX5000SetMotorCtrlWord.bForceUnLock XOR BreakUnlock)
																OR (SoEAX5000SetMotorCtrlWord.bForceLock XOR Breaklock)
																OR SoEAX5000SetMotorCtrlWord.bBusy;
END_METHOD

METHOD PUBLIC refreshStatus : BOOL //Return value = TRUE if busy
VAR_INPUT
END_VAR
IF __ISVALIDREF(rAxis) AND_THEN stateReadStatus = 0 
THEN
	stateReadStatus 										:= 10;
	StatusTrig.0 											:= rAxis.NcToPlc.StateDWord.28; (* DriveDeviceError *)
	StatusTrig.1 											:= rAxis.NcToPlc.StateDWord.30; (* IODataInvalid *)
	MEM_StatusTrig 											:= StatusTrig;
	MEMSET(ADR(DiagMsg),0,SIZEOF(DiagMsg));
	SoERead(bExecute := FALSE);
END_IF

RefreshStatus												:= stateReadStatus > 0;
END_METHOD

METHOD PUBLIC reset : BOOL //Return value = TRUE if busy
VAR_INPUT
END_VAR
reset													:= SoEDriveReset.bBusy OR NOT SoEDriveReset.bExecute;
SoEDriveReset.bExecute									:= NOT SoEDriveReset.bBusy AND NOT rAxis.Status.OpMode.SimulationAxis AND AdsAddr.port > 0;
END_METHOD

END_FUNCTION_BLOCK

// POUs/IO/Drives/SoE/AxDriveSoE_Ax5000CalcPower
FUNCTION_BLOCK AxDriveSoE_Ax5000CalcPower
VAR_INPUT
	Enable													:	BOOL;							// Enable functionblock
	ConfirmTrig												:	BOOL;							// Reset internal error
	ActParameterSet											:	INT := 0;						// Active arameter set of AX5000	Default := 0
END_VAR
VAR_IN_OUT	
(* important for function *)	
	AdsAddr													:	AMSADDR;						// AdsAddr of AX5000
	Channel													:	USINT;							// DriveChannel
END_VAR
VAR_OUTPUT
	AbsoluteVoltage								AT %I*		:	REAL;							// Need to be mapped!! Absolute Voltage read from parameter P-x-0469
	AbsoluteCurrent											:	REAL;							// Absolute Current calculated
	ActivePower												:	LREAL;							// Active power calculated in kW
	ReactivePower											:	LREAL;							// Reactive power calculated in kvar
	ApparentPower											:	LREAL;							// Apparent power calculated in kVA
	Busy													:	BOOL;							// Busy while SoeRead
	Error													:	BOOL;							// Error Bit
{attribute 'displaymode':='hex'}
	ErrorID													:	UDINT;							// ErrorID
	ErrorText												:	T_MaxString;					// ErrorText
END_VAR
VAR
	_AbsoluteCurrent							AT %I*		:	INT;		//	P-x-0461		// Need to be mapped!! Absolute Current: 1/1000% of PeakCurrent
(* Memory **********************************************************)
	State													:	INT;
	MemPeakCurrent											:	DINT;		//	P-x-0092		// Channel peak current, read from AX5000
	MemCosPhi												:	INT;		//	P-x-0104		// cos phi of motor, read from AX5000
	MemParamSet												:	INT := 99;
	
(* Functionsblocks *************************************************)
	rTrigExecute											:	R_TRIG;
	SoERead													:	FB_SoERead_ByDriveRef	:= (tTimeOut := DEFAULT_ADS_TIMEOUT);
(*******************************************************************)
END_VAR
VAR CONSTANT
	ST_IDLE													:	INT := 0;
	ST_PEAKCURRENT											:	INT := 10;
	ST_COSPHI												:	INT := 20;
	ST_ERROR												:	INT := 998;
	ST_RESET												:	INT := 999;
	
	ERR_PEAKCURRENT											:	UDINT := 1;
	ERR_COSPHI												:	UDINT := 2;
END_VAR


(* Init drive ref **************************************************)
	IF AdsAddr.port <> SoERead.stDriveRef.nSlaveAddr
	THEN
		SoERead.stDriveRef.sNetId							:= F_CreateAmsNetId(AdsAddr.netId);
		SoERead.stDriveRef.nSlaveAddr						:= AdsAddr.port;
		SoERead.stDriveRef.nDriveNo							:= Channel;
	END_IF
(* calculate  ******************************************************)
	IF NOT busy
		AND MemParamSet = ActParameterSet
		AND Enable
	THEN
		AbsoluteCurrent										:= TO_REAL(_AbsoluteCurrent * (MemPeakCurrent / 1000)) / 1000;
		ApparentPower										:= SQRT(3) * TO_LREAL(AbsoluteCurrent * AbsoluteVoltage)  / 1000;
		ActivePower											:= ApparentPower * TO_LREAL(MemCosPhi) / 100.0;
		ReactivePower										:= SQRT(EXPT(ApparentPower,2) - EXPT(ActivePower,2));
	END_IF
(* Trigger Execute *************************************************)
	rTrigExecute(CLK := MemParamSet <> ActParameterSet AND Enable);
	
(* get params ******************************************************)
	CASE state OF
	ST_IDLE:	
		IF rTrigExecute.Q
		THEN
			State											:= ST_PEAKCURRENT;
		END_IF
	ST_PEAKCURRENT:	// read P-x-0092 configured peak current
		IF NOT SoERead.bBusy
			AND SoERead.bExecute
		THEN
			state											:= SEL(SoERead.bError, ST_COSPHI, 99);
			ErrorID											:= SEL(SoERead.bError, 0, ERR_PEAKCURRENT);
			ErrorText										:= SEL(SoERead.bError, '', 'Fehler beim Lesen vom Kanal Spitzenstrom');
		END_IF
		SoERead(
			stDriveRef	:= ,  //See init for drive ref
			nIdn		:= Get_P_WORD(ActParameterSet) + 092,
			nElement	:= EC_SOE_ELEMENT_VALUE (* 16#40*),
			pDstBuf		:= ADR(MemPeakCurrent),
			cbBufLen	:= SIZEOF(MemPeakCurrent),
			bExecute	:= State = 10,
			tTimeout	:= ,
			bBusy		=> ,
			bError		=> ,
			iAdsErrId	=> ,
			iSercosErrId=> ,
			dwAttribute	=> );
	ST_COSPHI:	// read P-x-0104 cos phi
		IF NOT SoERead.bBusy
			AND SoERead.bExecute
		THEN
			MemParamSet										:= SEL(SoERead.bError, ActParameterSet, MemParamSet);
			state											:= SEL(SoERead.bError, ST_IDLE, ST_ERROR);
			ErrorID											:= SEL(SoERead.bError, 0, ERR_COSPHI);
			ErrorText										:= SEL(SoERead.bError, '', 'Fehler beim Lesen vom cos phi Parameter');
		END_IF
		SoERead(
			stDriveRef	:= ,  //See init for drive ref
			nIdn		:= Get_P_WORD(ActParameterSet) + 104,
			nElement	:= EC_SOE_ELEMENT_VALUE (* 16#40*),
			pDstBuf		:= ADR(MemCosPhi),
			cbBufLen	:= SIZEOF(MemCosPhi),
			bExecute	:= State = 20,
			tTimeout	:= ,
			bBusy		=> ,
			bError		=> ,
			iAdsErrId	=> ,
			iSercosErrId=> ,
			dwAttribute	=> );
	ST_ERROR:			// wait till Error is quit
		IF ConfirmTrig
		THEN
			ErrorText										:= '';
			ErrorID											:= 0;
			state											:= ST_RESET;
		END_IF
	ST_RESET:		
		IF NOT SoERead.bBusy
			AND NOT SoERead.bError
		THEN
			state											:= ST_IDLE;
		END_IF
		SoERead(
			stDriveRef	:= ,  //See init for drive ref
			nIdn		:= Get_P_WORD(ActParameterSet) + 092,
			nElement	:= EC_SOE_ELEMENT_VALUE (* 16#40*),
			pDstBuf		:= ADR(MemPeakCurrent),
			cbBufLen	:= SIZEOF(MemPeakCurrent),
			bExecute	:= FALSE,
			tTimeout	:= ,
			bBusy		=> ,
			bError		=> ,
			iAdsErrId	=> ,
			iSercosErrId=> ,
			dwAttribute	=> );
	END_CASE
	
	Error		:= state = ST_ERROR;
	Busy		:= state <> 0 OR SoERead.bBusy;
(*******************************************************************)

METHOD PRIVATE get_P_WORD : WORD
VAR_INPUT
	SetNumber			:	INT;
END_VAR
(* Get P-Word dependent of parameter set *)
	IF SetNumber = 0 THEN
		Get_p_WORD			:= P_0_IDN;
	ELSIF SetNumber = 1 THEN
		Get_P_WORD			:= P_1_IDN;
	ELSIF SetNumber = 2 THEN
		Get_P_WORD			:= P_2_IDN;
	ELSIF SetNumber = 3 THEN
		Get_P_WORD			:= P_3_IDN;
	ELSIF SetNumber = 4 THEN
		Get_P_WORD			:= P_4_IDN;
	ELSIF SetNumber = 5 THEN
		Get_P_WORD			:= P_5_IDN;
	ELSIF SetNumber = 6 THEN
		Get_P_WORD			:= P_6_IDN;
	ELSIF SetNumber = 7 THEN
		Get_P_WORD			:= P_7_IDN;
	END_IF
END_METHOD

METHOD PRIVATE get_S_WORD : WORD
VAR_INPUT
	SetNumber			:	INT;
END_VAR
(* Get S-Word dependent of parameter set *)
	IF SetNumber = 0 THEN
		Get_S_WORD			:= S_0_IDN;
	ELSIF SetNumber = 1 THEN
		Get_S_WORD			:= S_1_IDN;
	ELSIF SetNumber = 2 THEN
		Get_S_WORD			:= S_2_IDN;
	ELSIF SetNumber = 3 THEN
		Get_S_WORD			:= S_3_IDN;
	ELSIF SetNumber = 4 THEN
		Get_S_WORD			:= S_4_IDN;
	ELSIF SetNumber = 5 THEN
		Get_S_WORD			:= S_5_IDN;
	ELSIF SetNumber = 6 THEN
		Get_S_WORD			:= S_6_IDN;
	ELSIF SetNumber = 7 THEN
		Get_S_WORD			:= S_7_IDN;
	END_IF
END_METHOD

END_FUNCTION_BLOCK

// POUs/IO/Drives/SoE/AxDriveSoE_Ax5000Param
{attribute 'no_check'}
//FB template to read and write parameter
//The FB can be enherided and derivatived methods of SeqRead/SeqWrite used for application specific parameter.
//The extended methods need to call the super class at the beginning and return true if execution will be finished. The allowed states for new parameter are 1..99
FUNCTION_BLOCK AxDriveSoE_Ax5000Param EXTENDS AxRWParaBase
VAR_OUTPUT CONSTANT
END_VAR 
VAR_INPUT                               					
	AdsAddr													: 	AMSADDR; //Terminal AMS Net Addr. 
	Channel													:	USINT := 0; //Drive channel 0 or 1 for a two channel AX5000
	SetKvPosition											:	LREAL; //(rad/s)rad - e.g. 10.0		
	SetKpVelocity											:	LREAL; //mA/(rad/s) - e.g. 0.058	
	SetTnVelocity											:	LREAL; //0.1ms 		- e.g. 0.015	
END_VAR 
VAR_IN_OUT
END_VAR                               					
VAR_OUTPUT 	
//	MotorSN													:	STRING(15); 
	KvPosition												:	LREAL;
	KpVelocity												:	LREAL;
	TnVelocity												:	LREAL;	
	NominalMainVoltage										:	LREAL; //Volt                         										
	ErrorSoEId												:	UDINT := 0;
END_VAR                         	
VAR
(* Cache ************************************************************)

	
(* Trigger **********************************************************)

(* Timer ******************************************************************)

(* FBs ***************************************************************)
	SoEWrite												: 	FB_SoEWrite_ByDriveRef := (tTimeout := DEFAULT_ADS_TIMEOUT); //SoE read
	SoERead													: 	FB_SoERead_ByDriveRef := (tTimeout := DEFAULT_ADS_TIMEOUT); //SoE wriet

(* Dummy memory **********************************************************)

END_VAR

	(* Read/Write drive parameter														*)
	(************************************************************************************)
	
(* Execute ***************************************************************************************)
	SUPER^();
	
(*************************************************************************************************)

PROPERTY PROTECTED deviceAddrIsValid : BOOL
GET
deviceAddrIsValid := AdsAddr.port > 0;
END_GET
END_PROPERTY

METHOD PROTECTED getValue : BOOL //Return value = TRUE if execution finished and state incremented 
VAR_INPUT
	Idn							:	WORD;
	Element						:	BYTE;
	Len							:	UDINT;
	pActValue					:	PVOID; //Address of variable for actual value
	pSetValue					:	PVOID; //Address of variable for ser value variable, can be zero if no corresponding SetVariable exists
END_VAR

SoERead(bExecute := TRUE, nIdn := Idn, nElement := Element, pDstBuf := pActValue, cbBufLen := Len);
IF NOT SoERead.bBUSY 	
THEN
	IF NOT SoERead.bError
	THEN
		IF pSetValue <> 0 THEN MEMCPY(pSetValue, pActValue, Len); END_IF
		state 												:= state + 1; 
	ELSE
		Busy												:= FALSE;
		Error												:= TRUE;
		ErrorId												:= SoERead.iAdsErrId;
		ErrorSoEId											:= SoERead.iSercosErrId;
		ErrorText											:= CONCAT('Error read parameter in state:' , TO_STRING(state * -1));
		ErrorText											:= CONCAT(ErrorText , CONCAT(' Id:',TO_STRING(ErrorId)));
		ErrorText											:= CONCAT(ErrorText , CONCAT(' Sercos Err :',TO_STRING(ErrorSoEId)));
		State												:= 9999;
	END_IF
	SoERead(bExecute := FALSE);
	getValue												:= TRUE;
END_IF
END_METHOD

METHOD PROTECTED seqRead : BOOL //Return value = TRUE if execution finished 
VAR_IN_OUT
	State							:	INT;
END_VAR

(* Sequence read parameter **********************************)
	CASE state OF
	1..99: //Read application specific parameter  
		SeqRead												:= TRUE;
		
	1001: (* Init step ******************************************************)		
		SoERead(bExecute:=FALSE);
		IF NOT SoERead.bBusy
		THEN
			SoERead.stDriveRef.sNetId						:= F_CreateAmsNetId(AdsAddr.netId);	
			SoERead.stDriveRef.nSlaveAddr 					:= AdsAddr.port;
			SoERead.stDriveRef.nDriveNo 					:= TO_BYTE(Channel);			
			state											:= state + 1;	
		END_IF
		
	1002: (* Kv Position *************************************************************************************)
		IF getValue(Idn:= S_0_IDN + 104,	Element := EC_SOE_ELEMENT_VALUE,	LEN := SIZEOF(_UINT),		pActValue := ADR(_UINT),	pSetValue := 0 )
		THEN
			KvPosition	:= SetKvPosition					:= SEL(Error, TO_LREAL(_UINT) * 0.01, 0.0); 
		END_IF

	1003: (* Kp velocity *******************************************)
		IF getValue(Idn:= S_0_IDN + 100,	Element := EC_SOE_ELEMENT_VALUE,	LEN := SIZEOF(_UINT),		pActValue := ADR(_UINT),	pSetValue := 0 )
		THEN
			KpVelocity := SetKpVelocity						:= SEL(Error, TO_LREAL(_UDINT) * 0.001, 0.0);
		END_IF

	1004: (* Tn velocity ********************************************)
		IF getValue(Idn:= S_0_IDN + 101,	Element := EC_SOE_ELEMENT_VALUE,	LEN := SIZEOF(_UINT),		pActValue := ADR(_UINT),	pSetValue := 0 )
		THEN
			TnVelocity	:= SetTnVelocity					:= SEL(Error, TO_LREAL(_UINT) * 0.1, 0.0);
		END_IF
					
	1005: (* Nominal main voltage  ********************************************)
  		IF getValue(Idn:= P_0_IDN + 201,	Element := EC_SOE_ELEMENT_VALUE,	LEN := SIZEOF(_UINT),		pActValue := ADR(_UINT),	pSetValue := 0 )
		THEN
			NominalMainVoltage								:= SEL(Error, TO_LREAL(_UINT) * 0.1, 0.0);
		END_IF	
	ELSE
		state												:= 1;
	END_CASE

(***********************************************************************************)
END_METHOD

METHOD PROTECTED seqWrite : BOOL //Return value = TRUE if execution finished 
VAR_IN_OUT
	State							:	INT;
END_VAR
(* Sequence write parameter *********************************************)
	CASE state OF
	1..99: //Write application specific parameter  
		SeqWrite											:= TRUE;
		
	1001: (* Init step ******************************************************)		
		SoEWrite(bExecute:= TRUE);
		IF NOT SoEWrite.bBusy
		THEN
			SoEWrite.stDriveRef.sNetId						:= F_CreateAmsNetId(AdsAddr.netId);	
			SoEWrite.stDriveRef.nSlaveAddr 					:= AdsAddr.port;
			SoEWrite.stDriveRef.nDriveNo 					:= Channel;		
			state											:= state + 1;	
		END_IF
	
	1002: (* Kv position *************************************************************************************)
		_UINT												:= TO_UINT(SetKvPosition * 100.0);
		IF setValue(Idn := S_0_IDN + 104, Element := EC_SOE_ELEMENT_VALUE,	LEN := SIZEOF(_UINT),		pActValue := 0,		pSetValue := ADR(_UINT) )
		THEN
			KvPosition										:= SetKvPosition;
		END_IF		
		
	1003: (* Kp velocity ****************************************)
		_UDINT												:= TO_UDINT(SetKpVelocity * 1000.0);
		IF setValue(Idn := S_0_IDN + 100, Element := EC_SOE_ELEMENT_VALUE,	LEN := SIZEOF(_UDINT),		pActValue := 0,		pSetValue := ADR(_UDINT) )
		THEN
			KpVelocity										:= SetKpVelocity;
		END_IF	
		
	1004: (* Tn velocity **********************************)
		_UINT											:= TO_UINT(SetTnVelocity * 10.0);
		IF setValue(Idn := S_0_IDN + 101, Element := EC_SOE_ELEMENT_VALUE,	LEN := SIZEOF(_UINT),		pActValue := 0,		pSetValue := ADR(_UINT) )
		THEN
			TnVelocity										:= SetTnVelocity;
		END_IF		ELSE
		state												:= 1;
	END_CASE

(************************************************************************************)
END_METHOD

METHOD PROTECTED setValue : BOOL //Return value = TRUE if execution finished and state incremented 
VAR_INPUT
	Idn							:	WORD;
	Element						:	BYTE;
	Len							:	UDINT;
	pActValue					:	PVOID; //Address of variable for actual value, can be zero if no corresponding acual value variable exists
	pSetValue					:	PVOID; //Address of variable for set value variable
END_VAR

IF pActValue <> 0 AND pSetValue <> 0 AND_THEN MEMCMP(pSetValue, pActValue, Len) = 0
THEN //Skip write parameter if set and actual value are equel
	state													:= state + 1;	
	setValue												:= TRUE;
ELSE
	SoEWrite(bExecute:= TRUE, nIdn := Idn, nElement := Element, pSrcBuf := pSetValue, cbBufLen := LEN);
	IF NOT SoEWrite.bBusy
	THEN
		IF NOT SoEWrite.bError
		THEN
			IF pActValue <> 0 THEN MEMCPY(pActValue, pSetValue, Len); END_IF	
			state											:= state + 1;
		ELSE
			Busy											:= FALSE;
			Error											:= TRUE;
			ErrorId											:= SoEWrite.iAdsErrId;
			ErrorSoEId										:= SoEWrite.iSercosErrId;
			ErrorText										:= CONCAT('Error write parameter in state:' , TO_STRING(state * -1));
			ErrorText										:= CONCAT(ErrorText , CONCAT(' Id:',TO_STRING(ErrorId)));
			ErrorText										:= CONCAT(ErrorText , CONCAT(' Sercos Err :',TO_STRING(ErrorSoEId)));
			State											:= 9999;
		END_IF
		SoEWrite(bExecute := FALSE);
		setValue											:= TRUE;
	END_IF		
END_IF
END_METHOD

END_FUNCTION_BLOCK

// POUs/IO/Drives/SoE/AxDriveSoE_Ax5000SwitchParamSet
FUNCTION_BLOCK AxDriveSoE_Ax5000SwitchParamSet EXTENDS FbBase
VAR_INPUT
	rAxis													:	REFERENCE TO AXIS_REF := 0; 	// Axis Ref
	TimeOut													:	TIME := DEFAULT_ADS_TIMEOUT;	// Timeout time
	NewParamSet												:	INT;							// Value for new parameterset
END_VAR
VAR_IN_OUT	
(* important for function *)	
	AdsAddr													:	AMSADDR;						// AdsAddr of AX5000
	Channel													:	USINT;                          // Drive channel number
END_VAR
VAR_OUTPUT
	ErrorText												:	T_MaxString;					// Error Text
	ActParamSet												:	INT := -1; 						// Value of active parameter set
END_VAR
VAR
(* Memory **********************************************************)
	StartSwitchParamSet										:	INT := 0;
	
	CountError												:	USINT;
(* Timer ***********************************************************)
	TimerWait												:	TON;
	TimerTimeOut											:	TON;
	
(* Functionsblocks *************************************************)

	SoEWrite												:	FB_SoEWrite_ByDriveRef	:= (tTimeOut := DEFAULT_ADS_TIMEOUT);
	SoERead													:	FB_SoERead_ByDriveRef	:= (tTimeOut := DEFAULT_ADS_TIMEOUT);
(*******************************************************************)
END_VAR
VAR CONSTANT
	ST_IDLE													:	INT := 0;
	ST_REFRESH												:	INT := 10;
	ST_PRESELECT											:	INT := 100;
	ST_DISABLED												:	INT := 110;
	ST_RESETEXECUTE											:	INT := 120;
	ST_SETPARAM												:	INT := 130;
	ST_WAIT													:	INT := 140;
	ST_ERROR												:	INT := 998;
	ST_RESET												:	INT := 999;
	
	ERR_REFRESH												:	UDINT := 1;
	ERR_PRESELECT											:	UDINT := 2;
	ERR_TIMEOUT_DISABLED									:	UDINT := 3;
	ERR_RESETEXECUTE										:	UDINT := 4;
	ERR_EXECUTE												:	UDINT := 5;
	
	PT_WAIT_TIME											:	TIME := T#20MS;
END_VAR

(* abort function-call if the reference is invalid *****************)
	IF NOT __ISVALIDREF(rAxis) THEN
		Busy												:= NOT Error;
		Error												:= TRUE;
		ErrorId												:= 16#4B30;
		ErrorText											:= 'Referenz rAxis invalid (0)';
		RETURN;
	END_IF

(* Init drive ref **************************************************)
	IF AdsAddr.port <> SoERead.stDriveRef.nSlaveAddr
	THEN
		SoERead.stDriveRef.sNetId							:= F_CreateAmsNetId(AdsAddr.netId);
		SoERead.stDriveRef.nSlaveAddr						:= AdsAddr.port;
		SoERead.stDriveRef.nDriveNo							:= Channel;
		
		SoEWrite.stDriveRef									:= SoERead.stDriveRef;
	END_IF
(* Trigger Execute *************************************************)
	rtExecute(CLK := Execute);
	
(* switch parameter set ********************************************)
	CASE State OF
	ST_IDLE:			// wait for command
	(* Get actual parameter set after restart *)
		IF ActParamSet < 0 
		THEN
			State											:= ST_REFRESH;
	(* Start switch parameter set *)
		ELSIF rtExecute.Q
		THEN
			setNewParam(NewParamSet);
		ELSIF NOT Execute
		THEN
			Error											:= FALSE;
			Done											:= FALSE;
			Busy											:= TRUE;
			ErrorId											:= 0;
			ErrorTExt										:= '';
		END_IF
		
	ST_REFRESH: 		// Refresh ActParamSet Variable
		IF NOT SoERead.bBusy
			AND SoERead.bExecute
		THEN
			State											:= SEL(SoERead.bError, ST_IDLE, ST_ERROR);
			Done											:= State = ST_IDLE;
			Error											:= State = ST_ERROR;	
			ErrorID											:= SEL(SoERead.bError, 0, ERR_REFRESH);
			ErrorText										:= SEL(SoERead.bError, '', 'Fehler beim Aktualisieren des aktuellen Parametersatzes');
		END_IF
		
		SoERead(
			stDriveRef	:= ,  //See init for drive ref
			nIdn		:= S_0_IDN + 254,
			nElement	:= EC_SOE_ELEMENT_VALUE (* 16#40*),
			pDstBuf		:= ADR(ActParamSet),
			cbBufLen	:= SIZEOF(ActParamSet),
			bExecute	:= State = ST_REFRESH,
			tTimeout	:= ,
			bBusy		=> ,
			bError		=> ,
			iAdsErrId	=> ,
			iSercosErrId=> ,
			dwAttribute	=> );
			
		ST_PRESELECT:		// Set New param value in drive preselection
			IF NewParamSet = ActParamSet
			THEN
				State										:= ST_IDLE;
			ELSIF NOT SoEWrite.bBusy
				AND SoEWrite.bExecute
			THEN
				State										:= SEL(SoEWrite.bError, ST_DISABLED, ST_ERROR);
				ErrorID										:= SEL(SoERead.bError, 0, ERR_PRESELECT);
				ErrorText									:= SEL(SoERead.bError, '', 'Fehler beim Schreiben der Vorwahl');
			END_IF
			
			SoEWrite(
				stDriveRef	:= ,  //See init for drive ref
				nIdn		:= S_0_IDN + 217,
				nElement	:= EC_SOE_ELEMENT_VALUE (* 16#40*),
				pSrcBuf		:= ADR(NewParamSet),
				cbBufLen	:= SIZEOF(NewParamSet),
				bExecute	:= State = ST_PRESELECT,
				tTimeout	:= ,
				bBusy		=> ,
				bError		=> ,
				iAdsErrId	=> ,
				iSercosErrId=> );
				
		ST_DISABLED:		// check if axis is disabled
			TimerTimeOut(IN := NOT rAxis.Status.Disabled, PT := TimeOut);
			IF TimerTimeOut.Q THEN
				TimerTimeOut(IN := FALSE);
				State											:= ST_ERROR;
				ErrorID											:= SEL(SoERead.bError, 0, ERR_TIMEOUT_DISABLED);
				ErrorText										:= SEL(SoERead.bError, '', 'Achse ist nicht deaktiviert');
			ELSIF rAxis.Status.Disabled THEN
				TimerTimeOut(IN := FALSE);
				State											:= ST_RESETEXECUTE;
			END_IF
		
		ST_RESETEXECUTE:	// reset the execute command in drive	
			StartSwitchParamSet									:= 0;
			IF NOT SoEWrite.bBusy
				AND SoEWrite.bExecute
			THEN
				State											:= SEL(SoEWrite.bError, ST_SETPARAM, ST_ERROR);
				ErrorID											:= SEL(SoERead.bError, 0, ERR_RESETEXECUTE);
				ErrorText										:= SEL(SoERead.bError, '', 'Fehler beim Zurücksetzen des Ausführungskomamando');
			END_IF
			SoEWrite(
				stDriveRef	:= ,  //See init for drive ref
				nIdn		:= S_0_IDN + 216,
				nElement	:= EC_SOE_ELEMENT_VALUE (* 16#40*),
				pSrcBuf		:= ADR(StartSwitchParamSet),
				cbBufLen	:= SIZEOF(StartSwitchParamSet),
				bExecute	:= State = ST_RESETEXECUTE,
				tTimeout	:= ,
				bBusy		=> ,
				bError		=> ,
				iAdsErrId	=> ,
				iSercosErrId=> );		
				
		ST_SETPARAM:		// Execute switch parameter set
			StartSwitchParamSet								:= 3;
			IF NOT SoEWrite.bBusy
				AND SoEWrite.bExecute
			THEN
				State										:= SEL(SoEWrite.bError, ST_WAIT, ST_ERROR);
				ErrorID										:= SEL(SoERead.bError, 0, ERR_EXECUTE);
				ErrorText									:= SEL(SoERead.bError, '', 'Fehler beim Setzen des Ausführungskommandos');
			END_IF
			SoEWrite(
				stDriveRef	:= ,  //See init for drive ref
				nIdn		:= S_0_IDN + 216,
				nElement	:= EC_SOE_ELEMENT_VALUE (* 16#40*),
				pSrcBuf		:= ADR(StartSwitchParamSet),
				cbBufLen	:= SIZEOF(StartSwitchParamSet),
				bExecute	:= State = ST_SETPARAM,
				tTimeout	:= ,
				bBusy		=> ,
				bError		=> ,
				iAdsErrId	=> ,
				iSercosErrId=> );
				
		ST_WAIT:			// wait a short time while the drive works with the command
			TimerWait(IN := TRUE, pt := PT_WAIT_TIME);
			IF TimerWait.Q THEN
				TimerWait(IN := FALSE);
				State										:= ST_REFRESH;
			END_IF
			
		ST_ERROR:			// wait till Error is quit
			IF TRUE
			THEN
				State										:= ST_RESET;
			END_IF
			
		ST_RESET:			// Reset Error			
			State											:= ST_IDLE;
			SoEWrite(
				stDriveRef	:= ,  //See init for drive ref
				nIdn		:= S_0_IDN + 216,
				nElement	:= EC_SOE_ELEMENT_VALUE (* 16#40*),
				pSrcBuf		:= ADR(StartSwitchParamSet),
				cbBufLen	:= SIZEOF(StartSwitchParamSet),
				bExecute	:= FALSE,
				tTimeout	:= ,
				bBusy		=> ,
				bError		=> ,
				iAdsErrId	=> ,
				iSercosErrId=> );
			SoERead(
				stDriveRef	:= ,  //See init for drive ref
				nIdn		:= S_0_IDN + 254,
				nElement	:= EC_SOE_ELEMENT_VALUE (* 16#40*),
				pDstBuf		:= ADR(ActParamSet),
				cbBufLen	:= SIZEOF(ActParamSet),
				bExecute	:= FALSE,
				tTimeout	:= ,
				bBusy		=> ,
				bError		=> ,
				iAdsErrId	=> ,
				iSercosErrId=> ,
				dwAttribute	=> );
	END_CASE
	Busy													:= State <> ST_IDLE ;
(*******************************************************************)

METHOD setNewParam : BOOL	// Result = Busy
VAR_INPUT
	ParamNo					:	INT;
END_VAR

	IF ParamNo <> ActParamSet
		AND State = ST_IDLE
	THEN
		Error											:= FALSE;
		Done											:= FALSE;
		Busy											:= TRUE;
		ErrorId											:= 0;
		ErrorTExt										:= '';
		NewParamSet 									:= ParamNo;
		TimerWait(IN := FALSE);
		TimerTimeOut(IN := FALSE);
		State											:= ST_PRESELECT;
	END_IF
	
	SetNewParam											:= State <> ST_IDLE;
END_METHOD

END_FUNCTION_BLOCK

// POUs/IO/Drives/SoE/AxDriveSoE_Ax5000wEvents
{attribute 'no_check'}
//AX5000 SoE status and diagnosis FB with eventlogger 
FUNCTION_BLOCK AxDriveSoE_Ax5000wEvents EXTENDS AxDriveSoE_Ax5000
VAR_INPUT
	EnableEvent												:	BOOL := TRUE;
	ConfirmTrig												:	BOOL ;
	SourceId												:	UDINT := 102000; //SoE Drive default multisource Id + Ax id
	Name													:	STRING(30) := '';
	ErrorLimitPos											:	BOOL := FALSE;
	ErrorLimitNeg											:	BOOL := FALSE;
END_VAR                 									
VAR_IN_OUT              									
END_VAR                 									
VAR_OUTPUT              	                    										
	EventStatus												:	DWORD;
	NoOfActiveEvents										:	INT;
	Error													: 	BOOL; //ADS error SoE FBs
{attribute 'displaymode':='hex'}
	ErrorId													:	UDINT; //ADS error id of SoE FBs
	ErrorText												: 	STRING(40);
END_VAR
VAR_OUTPUT CONSTANT
END_VAR
VAR

(* Zwischenspeicher *********************************************************************)


(* Timer ********************************************************************************)

(* Trigger ******************************************************************************)

(* Bausteine ****************************************************************************)
	Event													:	EventHandlingGrp10;

(* Dummy Speicher **********************************************************)
	i														: INT := 0 ;


(****************************************************************************)
END_VAR

	(************************************************************************************)
	(*																					*)
	(*		B E C K H O F F   N E W   A U T O M A T I O N   T E C H N O L O G Y    		*)
	(*																					*)
	(*		Eiserstr.5	D-33415 Verl	Germany	phone:	+49-5246-0	www.Beckhoff.Com	*)
    (*																					*)
    (*		Bausteinbeschreibung	:	AX5000 Drive Ctrl								*)
	(*		TwinCAT-Version			:	3.x or higher 									*)
	(*		Version					:	V3.0 											*)
 	(*		Autor					:	Daniel Schlingmann								*)
	(*		Lib						:	TcMc2Drive.lib / TcDrive.Lib					*)
	(*																					*)
	(************************************************************************************)

(* Trigger reset if by active quit **********)
	IF ConfirmTrig
	THEN
		confirm();
	END_IF

(* Call super *****************************)
	SUPER^();
	
(* Call events ****************************************************)
	_callEvents();

(******************************************************************************)

METHOD PRIVATE _callEvents : BOOL
VAR_INPUT
END_VAR

(* Check if msg activ and init some parameter ***********************)
	IF Event.no[1].Text2 <> Name AND Name <> '' OR Event.no[1].Text2 = '' AND rAxis.NcToPlc.AxisId <> 0
	THEN
		Event.no[1].Class 									:= TC2_SYSTEM.TCEVENTCLASS_HINT;

		(* Init Name *)
		FOR i := Event.MIN_EVENT TO Event.MAX_EVENT DO
			Event.no[i].Text2								:= SEL(LEN(name)>1,CONCAT('Axis id:',DWORD_TO_STRING(rAxis.NcToPlc.AxisId)),name);
		END_FOR
	END_IF

(* workl Event Ctrl *************************************************)
	Event(
		ConfirmTrig := ConfirmTrig,
		Disable		:= rAxis.NcToPlc.AxisId = 0 OR NOT EnableEvent,
		SourceId	:= SourceId + rAxis.NcToPlc.AxisId,
		Status		=> EventStatus,
		NoOfActiveEvents => NoOfActiveEvents);

(* Error Hdl FB ******************************************************************)
	IF rAxis.Status.OpMode.SimulationAxis OR Event.confirmTrig
	THEN
		;
	ELSIF SoEDriveReset.bError
	THEN
		Error												:=	TRUE;
		ErrorId												:= 0;
		SercosErrorId										:= SoEDriveReset.iSercosErrId;
		ErrorText											:= CONCAT('SoeDrvReset SercosErrId: ',DWORD_TO_HEXSTR(SoEDriveReset.iSercosErrId,4,FALSE));
		ErrorText											:=	CONCAT(CONCAT(ErrorText,', ADSErrId: '),UINT_TO_STRING(SoEDriveReset.iAdsErrId));
	ELSIF SoEAX5000SetMotorCtrlWord.bError
	THEN
		Error												:=	TRUE;
		ErrorId												:= 0;
		SercosErrorId										:= SoEAX5000SetMotorCtrlWord.iSercosErrId;
		ErrorText											:= CONCAT('SoESetMotorCtrlWord SercosErrId: ',DWORD_TO_HEXSTR(SoEAX5000SetMotorCtrlWord.iSercosErrId,4,FALSE));
		ErrorText											:=	CONCAT(CONCAT(ErrorText,', ADSErrId: '),UINT_TO_STRING(SoEAX5000SetMotorCtrlWord.iAdsErrId));
	ELSIF SoERead.bError
	THEN
		Error												:=	TRUE;
		ErrorId												:= 0;
		SercosErrorId										:= SoERead.iSercosErrId;
		ErrorText											:= CONCAT('SoERead SercosErrId: ',DWORD_TO_HEXSTR(SoERead.iSercosErrId ,4,FALSE));
		ErrorText											:=	CONCAT(CONCAT(ErrorText,', ADSErrId: '),UINT_TO_STRING(SoERead.iAdsErrId));
	END_IF

(* Event Logger Meldungen *****************************************************)
	Event.no[1].Flag 										:= Status.bNotReadyToPowerUp;
	Event.no[2].Flag 										:= Status.bDrvShutdownBitC1D AND stateReadStatus = 0; Event.no[2].pText3 := ADR(DiagMsg.strData);
	Event.no[3].Flag 										:= FALSE;
	Event.no[4].Flag 										:= ErrorLimitPos;
	Event.no[5].Flag 										:= ErrorLimitNeg;
	Event.no[6].Flag 										:= SafetyError AND DiagNumber <> 16#0000_FDD9;
	Event.no[7].Flag 										:= FALSE;
	Event.no[8].Flag 										:= FALSE;
	Event.no[9].Flag 										:= FALSE;
	Event.no[10].Flag 										:= Error; Event.no[10].Text1 := TO_STRING(ErrorId);
	
(************************************************************************)
END_METHOD

METHOD PUBLIC confirm : BOOL //Return value = TRUE if busy
VAR_INPUT
END_VAR
Event.confirm();
Error												:= FALSE;
ErrorId												:= 0;
SercosErrorId										:= 0;
ErrorText											:= '';
		
confirm 											:= SUPER^.reset();
END_METHOD

END_FUNCTION_BLOCK

// POUs/IO/Drives/SoE/AxDriveSoE_Rexroth
{attribute 'no_check'}
//Bosch Rexroth EtherCAT SoE Drive Control
//based on Tc2_Drive
FUNCTION_BLOCK AxDriveSoE_Rexroth EXTENDS AxDriveBase
VAR_INPUT
	EnableEvent												:	BOOL := TRUE;
	ResetTrig												:	BOOL := FALSE; (* Quit event and reset drive (SoE Reset) *)
	SourceId												:	UDINT := 102000; //SoE Drive default multisource Id + Ax id
	Name													:	STRING(30) := '';
	ErrorLimitPos											:	BOOL := FALSE;
	ErrorLimitNeg											:	BOOL := FALSE;
	BreakUnlock												:	BOOL := FALSE; //Not implemented yet
	BreakLock												:	BOOL := FALSE; //Not implemented yet					
	SetReferenz												: 	BOOL := FALSE;
	Referenzpos												: 	LREAL := 0.0;
END_VAR                                 					
VAR_IN_OUT                              					
END_VAR                                 					
VAR_OUTPUT                                                					
	InReferenz												:	BOOL; (* Drive in reference *)
	RT_StatusChanged										:	BOOL;                                    						
	Status													:	ST_IndraDriveCsDriveStatus;
	C1D														:	ST_IndraDriveCs_C1D;
	DiagMsg 												: 	ST_SoE_String;
	DiagNumber 												: 	UDINT;
	Operational												: INPUT := (Force := TRUE);	(* Link to ALWAYS_TRUE or operational signal from drive *)
	EcState											AT %I* 	: 	UINT; (* Ethercat InfoData State *)
	SercosErrorId											:	UINT;                    					
	SafetyError										AT %I*	:	BOOL;	(* Ax5805 Drive Safety Error - Bit .7 in Input Safe Data Byte 0 oder 2 *)	
	EventStatus												:	DWORD;
	NoOfActiveEvents										:	INT;
	Busy													:	BOOL;
	Error													:	BOOL;
{attribute 'displaymode':='hex'}
	ErrorId													:	UDINT;
	ErrorText												:	STRING(40);
END_VAR                  						
VAR_OUTPUT CONSTANT
END_VAR
VAR (* EA Internal *)
	EcInfoDataState									AT %I* 	: 	UINT; (* Ethercat InfoData State *)
END_VAR
VAR

(* Cache *********************************************************************)
	MemDriveStatusword										: 	WORD;
	MEM_StatusTrig											:	BYTE;
	StatusTrig												:	BYTE;
	stateReadStatus											:	INT;
	stateCtrl												:	INT := 0;

(* Timer ********************************************************************************)

(* Trigger ******************************************************************************)

(* Instance ****************************************************************************)
	SoEDriveReset											: 	FB_SoEReset := (Timeout		:= DEFAULT_ADS_TIMEOUT);
	SoEWrite												: 	FB_SoEWrite := (Timeout		:= DEFAULT_ADS_TIMEOUT);
	SoERead													: 	FB_SoERead := (Timeout		:= DEFAULT_ADS_TIMEOUT);
	SoEExecuteCmd											:	FB_SoEExecuteCommand := (Timeout		:= DEFAULT_ADS_TIMEOUT);
	EcSetSlaveSTATE											:	FB_EcSetSlaveSTATE := (tTimeout		:= DEFAULT_ADS_TIMEOUT);
	Event													:	EventHandlingGrp10;

(* Dummy Speicher **********************************************************)
	i														: 	INT := 0 ;
	_word													:	WORD;
	_DWORD													:	DWORD;

(****************************************************************************)
END_VAR

	(************************************************************************************)
	(*																					*)
	(*		B E C K H O F F   N E W   A U T O M A T I O N   T E C H N O L O G Y    		*)
	(*																					*)
	(*		Eiserstr.5	D-33415 Verl	Germany	phone:	+49-5246-0	www.Beckhoff.Com	*)
    (*																					*)
    (*		Bausteinbeschreibung	:	Ethercat SoE MC2 Drive Ctrl						*)
	(*		TwinCAT-Version			:	3.x or higher	 								*)
	(*		Version					:	V3.0/05/11										*)
 	(*		Autor					:	Daniel Schlingmann								*)
	(*		Lib						:	TcMC2Drive.lib / TcDrive.Lib					*)
	(*																					*)
	(* Call cyclic																		*)
	(************************************************************************************)

(* abort function-call if the reference is invalid *****************************)
IF NOT __ISVALIDREF(rAxis)  
THEN
	Busy													:= NOT Error;
	Fault													:= TRUE;
	Ready													:= FALSE;
	Error													:= TRUE;
	ErrorId													:= 16#4B30;
	ErrorText												:= 'Referenz rAxis invalid (0)';
	SercosErrorId											:= 0;
	RETURN;
END_IF

(* DriveStatusword *****************************)
	Status 													:= F_ConvWordToSTIndraDriveCsDriveStatus(StatusWord);
	IF rAxis.Status.OpMode.SimulationAxis or AdsAddr.port = 0
	THEN
		Status.bNotReadyToPowerUp							:= FALSE;	
		Status.bDrvShutdownBitC1D							:= FALSE;
		Status.bReadyForEnable								:= TRUE;
		Status.bEnabled										:= TRUE;	
	END_IF
	
(* Drive Operation Input ***********************)
	Operational(
		Force		:= rAxis.Status.OpMode.SimulationAxis ,
		Invert		:= ,
		PT_ON		:= ,
		PT_OFF		:= ,
		Q_DIRECT	=> ,
		Q			=> ,
		Q_RT		=> ,
		Q_FT		=> );

(* DriveStatusBits ***********************************************)
	Fault													:= Status.bDrvShutdownBitC1D
																OR rAxis.NcToPlc.StateDWord.28 (* DriveDeviceError *)
																OR rAxis.NcToPlc.StateDWord.30; (* IODataInvalid *)
                                						
	Ready 													:= NOT Fault
																	AND(Status.bReadyForEnable OR Status.bEnabled)
																	AND Operational.Q;
  
	SwitchedOn												:= Status.bEnabled AND NOT Fault;	
	                              	
(* Reset Drive ****************************************************)
	SoEDriveReset(
		NetId		:= ,
		Execute		:= ,
		Timeout		:= ,
		Axis		:= rAxis,
		Busy		=> ,
		Error		=> ,
		AdsErrId	=> ,
		SercosErrId	=> );

	IF SoEDriveReset.Busy 
	THEN
		; (* Block ist currend working *)
	ELSIF ResetTrig
	THEN
		reset();
	ELSIF SoEDriveReset.Execute
	THEN
	(*	RefreshStatus();  *)
		SoEDriveReset.Execute 								:= FALSE;
	END_IF

(* Set Etehrcat State to OP ********************************************)
	EcSetSlaveSTATE(
		sNetId		:= F_CreateAmsNetId(nIds := AdsAddr.netId),
		nSlaveAddr	:= AdsAddr.port,
		bExecute	:= ,
		tTimeout	:= ,
		reqState	:= Tc2_EtherCAT.EC_DEVICE_STATE_OP,
		bBusy		=> ,
		bError		=> ,
		nErrId		=> ,
		currState	=> );

	IF EcSetSlaveSTATE.bBusy
	THEN
		; (* Block ist currend working *)
	ELSIF EcSetSlaveSTATE.bExecute
		AND NOT ResetTrig
	THEN
		RefreshStatus();
		EcSetSlaveSTATE.bExecute 							:= FALSE;
	END_IF

(* Referenzieren *******************************************************)
	CASE stateCtrl OF
	-1,0:
		IF SetReferenz AND NOT rAxis.Status.OpMode.SimulationAxis AND AdsAddr.port > 0
		THEN
			writeReferenz();
		ELSE
			stateCtrl										:= 0;
		END_IF

	1: (* Referezwert schreiben **************************************)
		IF NOT SoEWrite.Busy
			AND SoEWrite.Execute
		THEN
			IF SoEWrite.Error
			THEN
				stateCtrl 									:= 0;
			ELSE                							
				stateCtrl									:= 2;
			END_IF
		END_IF

		_DWORD 												:= LREAL_TO_UDINT(Referenzpos);

		SoEWrite(
			NetId		:= ,
			Idn			:= S_0_IDN + 52,
			Element		:= EC_SOE_ELEMENT_VALUE ,
			pSrcBuf		:= ADR(_DWORD),
			BufLen		:= SIZEOF(_DWORD),
			Execute		:= stateCtrl = 1,
			Timeout		:= ,
			Password	:= ,
			Axis		:= rAxis,
			Busy		=> ,
			Error		=> ,
			AdsErrId	=> ,
			SercosErrId	=> );

	2: (* commad for setting setvalue *)
		IF NOT SoEExecuteCmd.Busy
			AND SoEExecuteCmd.Execute
		THEN
			IF SoEExecuteCmd.Error
			THEN
				stateCtrl 									:= 0;
			ELSE
				RefreshStatus();
				IF NOT SetReferenz
				THEN
					stateCtrl 								:= 0;
				ELSE            							
					stateCtrl 								:= -1;
				END_IF
			END_IF
		END_IF

		SoEExecuteCmd(
			NetId		:= '',
			Idn			:= P_0_IDN + 12,
			Execute		:= stateCtrl = 2,
			Timeout		:= ,
			Axis		:= rAxis,
			Busy		=> ,
			Error		=> ,
			AdsErrId	=> ,
			SercosErrId	=> );
	ELSE
		;
	END_CASE


(* evaluate sercos DriveStatusword *********************************************************)
	RT_StatusChanged 										:= SHR(StatusWord,2) <> MemDriveStatusword;
	MemDriveStatusword 										:= SHR(StatusWord,2);

(* Start Read Drive status *****************************************************************)
	CASE stateReadStatus OF
	0:
		StatusTrig.0 										:= rAxis.NcToPlc.StateDWord.28; (* DriveDeviceError *)
		StatusTrig.1 										:= rAxis.NcToPlc.StateDWord.30; (* IODataInvalid *)
                                							
		IF NOT rAxis.Status.OpMode.SimulationAxis AND AdsAddr.port > 0
			AND(RT_StatusChanged OR MEM_StatusTrig <> StatusTrig)
		THEN
			RefreshStatus();
		ELSE
			;
		END_IF

	(* Read Class 1 Diag *********************************************************)
	10:
		IF NOT SoERead.Busy
			AND SoERead.Execute
		THEN
			IF SoERead.Error
			THEN
				stateReadStatus 							:= 0;
			ELSE                    						
				C1D 										:= F_ConvWordToSTIndraDriveCsC1D(_word);
				stateReadStatus 							:= stateReadStatus + 1;
			END_IF
		END_IF

		SoERead(
			NetId		:= ,
			Idn			:= S_0_IDN + 11,
			Element		:= EC_SOE_ELEMENT_VALUE,
			pDstBuf		:= ADR(_word),
			BufLen		:= SIZEOF(_word),
			Execute		:= stateReadStatus = 10,
			Timeout		:= ,
			Axis		:= rAxis,
			Busy		=> ,
			Error		=> ,
			AdsErrId	=> ,
			SercosErrId	=> ,
			Attribute	=> );

	(* S-0-0403 In Referenz ********************************************************)
	11:
		IF NOT SoERead.Busy
			AND SoERead.Execute
		THEN
			IF SoERead.Error
			THEN
				stateReadStatus 							:= 0;
			ELSE
				InReferenz 									:= _WORD.0 AND _WORD.1;
				stateReadStatus 							:= stateReadStatus + 1;
			END_IF
		END_IF

		SoERead(
			NetId		:= ,
			Idn			:= S_0_IDN + 403,
			Element		:= EC_SOE_ELEMENT_VALUE,
			pDstBuf		:= ADR(_word),
			BufLen		:= SIZEOF(_word),
			Execute		:= stateReadStatus = 11,
			Timeout		:= ,
			Axis		:= rAxis,
			Busy		=> ,
			Error		=> ,
			AdsErrId	=> ,
			SercosErrId	=> ,
			Attribute	=> );

			
	(* Diag Message *********************************************************)
	12:
		IF NOT SoERead.Busy
			AND SoERead.Execute
		THEN
			IF SoERead.Error
			THEN
				stateReadStatus 							:= 0;
			ELSE
				stateReadStatus 							:= stateReadStatus + 1;
			END_IF
		END_IF

		SoERead(
			NetId		:= ,
			Idn			:= S_0_IDN + 95,
			Element		:= EC_SOE_ELEMENT_VALUE (* 16#40*),
			pDstBuf		:= ADR(DiagMsg),
			BufLen		:= SIZEOF(DiagMsg),
			Execute		:= stateReadStatus = 12,
			Timeout		:= ,
			Axis		:= rAxis,
			Busy		=> ,
			Error		=> ,
			AdsErrId	=> ,
			SercosErrId	=> ,
			Attribute	=> );

	(* Diag Number *********************************************************)
	13:
		IF NOT SoERead.Busy
			AND SoERead.Execute
		THEN
			IF SoERead.Error
			THEN
				stateReadStatus 							:= 0;
			ELSE
				stateReadStatus 							:= stateReadStatus + 1;
			END_IF
		END_IF

		SoERead(
			NetId		:= ,
			Idn			:= S_0_IDN + 390,
			Element		:= EC_SOE_ELEMENT_VALUE (* 16#40*),
			pDstBuf		:= ADR(DiagNumber),
			BufLen		:= SIZEOF(DiagNumber),
			Execute		:= stateReadStatus = 13,
			Timeout		:= ,
			Axis		:= rAxis,
			Busy		=> ,
			Error		=> ,
			AdsErrId	=> ,
			SercosErrId	=> ,
			Attribute	=> );
			
	(* reading status finished ************************************************************)
	ELSE (* Case else *)
		stateReadStatus 									:= 0;
	END_CASE

(* Event Logger Meldungen *****************************************************)
	Event.no[1].Flag 										:= Status.bNotReadyToPowerUp;
	Event.no[2].Flag 										:= Status.bDrvShutdownBitC1D AND stateReadStatus = 0; Event.no[2].pText3 := ADR(DiagMsg.strData);
	Event.no[3].Flag 										:= FALSE;
	Event.no[4].Flag 										:= ErrorLimitPos;
	Event.no[5].Flag 										:= ErrorLimitNeg;
	Event.no[6].Flag 										:= FALSE; //SafetyError AND DiagNumber <> 16#0000_FDD9;
	Event.no[7].Flag 										:= FALSE;
	Event.no[8].Flag 										:= FALSE;
	Event.no[9].Flag 										:= FALSE;
	Event.no[10].Flag 										:= Error;

	(* Check if msg activ and init some parameter ***********************)
	IF Event.no[1].Text2 <> Name AND Name <> '' OR Event.no[1].Text2 = '' AND rAxis.NcToPlc.AxisId <> 0
	THEN
		Event.no[1].Class 									:= TC2_SYSTEM.TCEVENTCLASS_HINT;

		(* Init Name *)
		FOR i := Event.MIN_EVENT TO Event.MAX_EVENT DO
			Event.no[i].Text2								:= SEL(LEN(name)>1,CONCAT('Axis id:',DWORD_TO_STRING(rAxis.NcToPlc.AxisId)),name);
		END_FOR
	END_IF

(* workl Event Ctrl *************************************************)
	Event(
		ConfirmTrig := ResetTrig,
		Disable		:= rAxis.NcToPlc.AxisId = 0 OR NOT EnableEvent,
		SourceId	:= SourceId + rAxis.NcToPlc.AxisId,
		Status		=> EventStatus,
		NoOfActiveEvents => NoOfActiveEvents);
				
(* Error Hdl FB ******************************************************************)
	IF SoEDriveReset.Error
	THEN
		Error												:=	TRUE;
		ErrorId												:= 0;
		SercosErrorId										:= SoEDriveReset.SercosErrId;
		ErrorText											:= CONCAT('SoeDrvReset SercosErrId: ',DWORD_TO_HEXSTR(SoEDriveReset.SercosErrId,4,FALSE));
		ErrorText											:=	CONCAT(CONCAT(ErrorText,', ADSErrId: '),UINT_TO_STRING(SoEDriveReset.AdsErrId));
	ELSIF SoEExecuteCmd.Error
	THEN
		Error												:=	TRUE;
		ErrorId												:= 0;
		SercosErrorId										:= SoEExecuteCmd.SercosErrId;
		ErrorText											:= CONCAT('SoEExecuteCmd SercosErrId: ',DWORD_TO_HEXSTR(SoEExecuteCmd.SercosErrId,4,FALSE));
		ErrorText											:=	CONCAT(CONCAT(ErrorText,', ADSErrId: '),UINT_TO_STRING(SoEExecuteCmd.AdsErrId));
	ELSIF SoERead.Error
	THEN
		Error												:=	TRUE;
		ErrorId												:= 0;
		SercosErrorId										:= SoERead.SercosErrId;
		ErrorText											:= CONCAT('SoERead SercosErrId: ',DWORD_TO_HEXSTR(SoERead.SercosErrId,4,FALSE));
		ErrorText											:=	CONCAT(CONCAT(ErrorText,', ADSErrId: '),UINT_TO_STRING(SoERead.AdsErrId));
	ELSIF SoEWrite.Error
	THEN
		Error												:=	TRUE;
		ErrorId												:= 0;
		SercosErrorId										:= SoEWrite.SercosErrId;
		ErrorText											:= CONCAT('SoEWrite SercosErrId: ',DWORD_TO_HEXSTR(SoEWrite.SercosErrId,4,FALSE));
		ErrorText											:=	CONCAT(CONCAT(ErrorText,', ADSErrId: '),UINT_TO_STRING(SoEWrite.AdsErrId));
	END_IF

(* FB is Busy *******************************************************************)
	Busy 													:= stateCtrl > 0
																OR SoEDriveReset.Busy
																OR stateReadStatus > 0;

(******************************************************************************)

METHOD PUBLIC refreshStatus : BOOL //Return value = TRUE if busy
VAR_INPUT
END_VAR
IF NOT __ISVALIDREF(rAxis)  
THEN
	Busy													:= NOT Error;
	Error													:= TRUE;
	ErrorId													:= 16#4B30;
	ErrorText												:= 'Referenz rAxis invalid (0)';
	SercosErrorId											:= 0;
ELSIF stateReadStatus = 0 
THEN
	Busy													:= TRUE;
	Error													:= FALSE;
	ErrorTExt												:= '';
	ErrorId													:= 0;
	SercosErrorId											:= 0;
	stateReadStatus 										:= 10;
	StatusTrig.0 											:= rAxis.NcToPlc.StateDWord.28; (* DriveDeviceError *)
	StatusTrig.1 											:= rAxis.NcToPlc.StateDWord.30; (* IODataInvalid *)
	MEM_StatusTrig 											:= StatusTrig;
	MEMSET(ADR(DiagMsg),0,SIZEOF(DiagMsg));
	SoERead(
		Execute := FALSE,
		Axis 	:= rAxis);
ELSE
	Busy													:= TRUE;
END_IF                              						
                                    						
RefreshStatus												:= Busy AND stateReadStatus > 0;
END_METHOD

METHOD PUBLIC reset : BOOL //Return value = TRUE if busy
VAR_INPUT
END_VAR
IF NOT SoEDriveReset.Execute
THEN
	Error													:=	FALSE;
	ErrorId													:= 0;
	SercosErrorId											:= 0;
	Errortext												:= '';
END_IF
EcSetSlaveSTATE.bExecute									:= NOT (( UINT_TO_WORD(EcState) AND Tc2_EtherCAT.EC_DEVICE_STATE_MASK ) = Tc2_EtherCAT.EC_DEVICE_STATE_OP)
																AND EcState > 0 AND NOT rAxis.Status.OpMode.SimulationAxis;
										
Busy														:= SoEDriveReset.Busy OR NOT SoEDriveReset.Execute;               							
SoEDriveReset.Execute										:= NOT SoEDriveReset.Busy AND NOT rAxis.Status.OpMode.SimulationAxis AND AdsAddr.port > 0;
reset													:= Busy;
END_METHOD

METHOD PUBLIC writeReferenz : BOOL //Return value = TRUE if busy
VAR_INPUT
END_VAR
IF NOT __ISVALIDREF(rAxis)  
THEN
	Busy													:= NOT Error;
	Error													:= TRUE;
	ErrorId													:= E_AdsErr.DEVICE_INVALIDPARM;
	ErrorText												:= 'Referenz rAxis invalid (0)';
	SercosErrorId											:= 0;
ELSIF stateCtrl = 0 
THEN
	ErrorText												:= '';
	Error													:=	FALSE;
	ErrorId													:= 0;
	SercosErrorId											:= 0;
	Busy													:= TRUE;
	stateCtrl 												:= 1;
	SoEWrite(Execute := FALSE, Axis := rAxis);
	SoEExecuteCmd(Execute := FALSE, Axis := rAxis);

END_IF                              						
                                    	
writeReferenz													:= Busy AND stateCtrl > 0;
END_METHOD

END_FUNCTION_BLOCK

// POUs/IO/Drives/Stepper/AxDriveStepper_wEvents
{attribute 'no_check'}
//Beckhoff Stepper terminal diag and diagnosis with eventlogger - extended from AxDriveStepper
//EventHandling instance use inside
FUNCTION_BLOCK AxDriveStepper_wEvents EXTENDS AxDriveStepper
VAR CONSTANT         	
END_VAR  
VAR_INPUT
	EnableEvent												:	BOOL := TRUE; //Enable to show events
	ConfirmTrig												:	BOOL := FALSE; //Quit events
	SourceId												:	UDINT := 102600; //MDP742 Stepper CoE Drive default multisource Id + Ax id
	Name													:	STRING(30) := '';
	ErrorLimitPos											:	BOOL := FALSE;
	ErrorLimitNeg											:	BOOL := FALSE;
END_VAR                     					
VAR_IN_OUT                  					
END_VAR                     					
VAR_OUTPUT                  					
 	EventStatus												:	DWORD;       
	NoOfActiveEvents										:	INT;                    					
END_VAR                     					                   					
VAR                         					
END_VAR
VAR

(* Cache *********************************************************************)
	
(* Timer ********************************************************************************)

(* Trigger ******************************************************************************)

(* Instance ****************************************************************************)
	Event													:	EventHandlingGrp10;
	
(* Dummy Speicher **********************************************************)
	i														: INT := 0 ;
END_VAR

	(* Stepper Drive Control with events												*)
	(************************************************************************************)

(* Call super **********************************************)
	SUPER^();
	
(* work events *******************************************)
	_callEvents();

(*******************************************************)

METHOD PRIVATE _callEvents : BOOL
VAR_INPUT
END_VAR

(* Check if msg activ and init some parameter ***********************)
	IF Event.no[1].Text2 <> Name AND Name <> '' OR Event.no[1].Text2 = '' AND rAxis.NcToPlc.AxisId <> 0
	THEN
		Event.no[1].Class 									:= TC2_SYSTEM.TCEVENTCLASS_STATEINFO;
		Event.no[3].Class 									:= TC2_SYSTEM.TCEVENTCLASS_MESSAGE;
		
		(* Init Achsname *)
		FOR i := Event.MIN_EVENT TO Event.MAX_EVENT DO
		(*	Event.no[i].Text1								:= '';*)
			Event.no[i].Text2								:= SEL(LEN(name)>1,CONCAT('Axis id:',DWORD_TO_STRING(rAxis.NcToPlc.AxisId)),name);
		END_FOR
	END_IF

(* workl Event Ctrl *************************************************)
	Event(
		ConfirmTrig := ConfirmTrig,
		Disable		:= rAxis.NcToPlc.AxisId = 0 OR NOT EnableEvent,
		SourceId	:= SourceId + rAxis.NcToPlc.AxisId,
		Status		=> EventStatus,
		NoOfActiveEvents => NoOfActiveEvents);

(* Event Logger Meldungen *****************************************************)
	Event.no[1].Flag 										:= NOT Status_ReadyToEnable ; 
	Event.no[2].Flag 										:= Fault;
	Event.no[3].Flag 										:= (Status_Warning OR Diag_Configuration) AND NOT rAxis.Status.Homing AND rAxis.Status.Operational; //Avoid warning if drive is disabled (EL7037 and older FW on EL7047 <=06 - 2020-03-26) 				
	Event.no[4].Flag 										:= Diag_TorqueOverloaded;
	Event.no[5].Flag 										:= Diag_UnderVoltage OR Diag_OverVoltage OR Diag_NoControlPower;
	Event.no[6].Flag 										:= Diag_ShortCircuit OR Diag_ShortCircuitB OR Diag_OpenLoadA OR Diag_OpenLoadB; 
	Event.no[7].Flag 										:= Diag_Saturated;
	Event.no[8].Flag										:= Diag_OverTemperature ;
	Event.no[9].Flag 										:= ErrorLimitPos; 	
	Event.no[10].Flag 										:= ErrorLimitNeg;	
(*	Event.no[11].Flag 										:= FALSE; 				
	Event.no[12].Flag 										:= FALSE;					
	Event.no[13].Flag 										:= FALSE; 			Event.no[9].Class := TC2_SYSTEM.TCEVENTCLASS_WARNING;
	Event.no[14].Flag 										:= FALSE; 			Event.no[10].Class := TC2_SYSTEM.TCEVENTCLASS_WARNING;
	Event.no[15].Flag 										:= FALSE;
	Event.no[16].Flag 										:= FALSE;
	Event.no[17].Flag 										:= FALSE;
	Event.no[18].Flag 										:= FALSE;
	Event.no[19].Flag 										:= FALSE;
	Event.no[20].Flag 										:= FALSE;
	Event.no[21].Flag 										:= FALSE;
	Event.no[22].Flag 										:= FALSE;
	Event.no[23].Flag 										:= FALSE;
	Event.no[24].Flag 										:= FALSE;
	Event.no[25].Flag 										:= FALSE;
*)

(******************************************************************************)
END_METHOD

METHOD PUBLIC confirm : bool
VAR_INPUT
END_VAR
confirm			:= Event.confirm();
END_METHOD

END_FUNCTION_BLOCK

// POUs/IO/Drives/Stepper/AxDriveStepperParam
{attribute 'no_check'}
//FB template to read and write parameter
//The FB can be enherided and derivatived methods of SeqRead/SeqWrite used for application specific parameter.
//The extended methods need to call the super class at the beginning and return true if execution will be finished. The allowed states for new parameter are 1..99
//
//Calculating NC-parameter
//Sacling with Enc 		= Distance per revolution / (Increments x 4 fold)
//Scaling without Enc.  = Distance per revolution / (Fullsteps x Microsteps)
//Scalingfactor = 360° / (1024 x 4) OR 360° / (200 x 64) 
//
//Ref. Velocity = (Max. Outputfreq * Distance per rev.) / (Fullsteps * Microsteps)
//3515 °/s = (126kHz * 360°) / (200 * 64)
//Set kv to 0 to see whether ref. velocity is correct
//
FUNCTION_BLOCK AxDriveStepperParam EXTENDS AxRWParaBase
VAR_OUTPUT CONSTANT
END_VAR                                 					
VAR_INPUT                               					
	AdsAddr													: 	AMSADDR; //Terminal AMS Net Addr.                                        	                                        	
	Channel													:	USINT := 0; //Drive channel 0 or 1 
	SetKpPosition											:	LREAL; //0:8014:02 - only at EL70x7
	SetKpVelocity											:	LREAL; //0:8014:03 in 0.1mA/(rad/s) - at EL70x1 -> 0:8013:01 - at EL70x1
	SetKiVelocity											:	LREAL; //0:8013:02 in 0.001 - NOT for EL70x7
	SetTnVelocity											:	LREAL; //0:8014:04 in 0.01 ms - only at EL70x7 
	SetKpCurrent											:	LREAL; //0:8011:01 
	SetKiCurrent											:	LREAL; //0:8011:02 

	SetCalibrInvertDirForCamSearch							:	BOOL; 	//0:8021:13 / TRUE=Cam search direction negative
	SetCalibrInvertDirForOfCam								:	BOOL; 	//0:8021:14 / TRUE=Sync impuls (off cam) search direction negative
	SetCalibrPosition										:	UDINT;	//0:8020:08 
END_VAR 
VAR_IN_OUT
END_VAR                               					
VAR_OUTPUT
	DeviceType												:	STRING(15); //e.g. EL7037

	KpPosition												:	LREAL;
	KpVelocity												:	LREAL;
	KiVelocity												:	LREAL; //Not available at EL70x7
	TnVelocity												:	LREAL; //Only available at EL70x7
	KpCurrent												:	LREAL;
	KiCurrent												:	LREAL;	
	CalibrInvertDirForCamSearch								:	BOOL; // TRUE=Cam search direction negative
	CalibrInvertDirForOfCam									:	BOOL; // TRUE=Sync impuls (off cam) search direction negative
	CalibrPosition											:	UDINT;
END_VAR                         	
VAR
(* Cache ************************************************************)
	
(* Trigger **********************************************************)

(* Timer ******************************************************************)

(* FBs ***************************************************************)
	CoEWrite												: FB_EcCoESdoWriteEx := (tTimeout := DEFAULT_ADS_TIMEOUT);
	CoERead													: FB_EcCoeSdoReadEx := (tTimeout := DEFAULT_ADS_TIMEOUT);

(* Dummy memory **********************************************************)
END_VAR

	(* Read/Write stepper drive parameter												*)
	(************************************************************************************)

(* Execute ***************************************************************************************)
	SUPER^();
	
(*************************************************************************************************)

PROPERTY PROTECTED deviceAddrIsValid : BOOL
GET
deviceAddrIsValid := AdsAddr.port > 0;
END_GET
END_PROPERTY

